// SIMATIC STEP 7 (V5.x) project 1300
// CPU: CPU 315-2 DP
// station: P_ADR_BUS
// station: Hardware
// station: SIMATIC 300(1)
// program: S7 Program(1)

SYMBOL_TABLE
"CLOCK_OP"	DB 5	DB 5	// COMMUNICATION CLOCK OP
"TransferValves"	DB 10	DB 10	// Data Transfer for Valves
"TransferMotor"	DB 11	DB 11	// Data Transfer for Motor
"TransferLevel"	DB 12	DB 12	// Data Transfer for Level
"TransferPressure"	DB 13	DB 13	// Data Transfer for Pressure
"TransferTemperature"	DB 14	DB 14	// Data Transfer for Temperatuer
"TransferPID"	DB 15	DB 15	// Data Transfer for PID
"TransferFlow"	DB 16	DB 16	// Data Transfer for Flow
"TrasferViskosity"	DB 17	DB 17	// Data Transfer for Viskosity
"TransferWeight"	DB 18	DB 18	// Data Transfer for Weight
"TransferGenerell"	DB 30	DB 30	// Data Transfer Generell
"Instance_FC_9_00"	DB 50	FB 110	// Instancename
"Instance_TC_10_01"	DB 51	FB 110	// Instance TC 10.01
"TransferRecipe"	DB 90	DB 90	// Data Transfer fo Recipe
"TransferBatch"	DB 91	DB 91
"DataBatchStarch"	DB 92	FB 90
"DataBatchCaCO3"	DB 93	FB 90
"ALARMTIME"	DB 100	DB 100	// actual timers alarms
"ALARMBLOCK"	DB 110	DB 110	// alarm indication to OP
"ALARM_ACK_OP"	DB 115	DB 115	// alarm acknowledge from OP
"LAMPS_ACK"	DB 120	DB 120	// lamp acknowledge
"CLOCK_FB"	FB 5	FB 5	// SETTING CPU CLOCK
"preparation starch"	FB 10	FB 10	// starch preparation
"starch cooking"	FB 11	FB 11	// starch jet cooker
"preparation CaCO3"	FB 15	FB 15	// CaCO3 preparation
"Devices"	FB 20	FB 20	// Devices
"ALARM_HANDLING_STARCH"	FB 31	FB 31	// alarm handling starch
"ALARM_HANDLING_CaCO3"	FB 32	FB 32	// alarm handling CaCO3
"ALARM"	FB 33	FB 33	// indication alarm
"CONT_C"	FB 41	FB 41	// Continuous Control
"Batch"	FB 90	FB 90	// Batch
"Control"	FB 110	FB 110	// Controler
"BatchControlStarch"	FC 10	FC 10	// Batch Control Starch
"BatchControlCaCO3"	FC 11	FC 11	// Batch Control CaCO3
"Recipe Control"	FC 90	FC 90	// Recipe Control
"DosLine"	FC 91	FC 91	// Dosing Line
"AUTO_VALVE"	FC 100	FC 100	// automatic valve
"MOTOR"	FC 101	FC 101	// motor control
"level"	FC 107	FC 107	// level display
"temperature"	FC 109	FC 109	// temperature display
"flow"	FC 110	FC 110	// flow display
"AI_4-20"	FC 111	FC 111	// analog input 4-20mA
"AO_4-20"	FC 112	FC 112	// analog output 4-20mA
"weight"	FC 114	FC 114	// weighing unit
"ALARM_BLOCK"	FC 115	FC 115	// alarm function block
"M2_01_RUN"	I 8.0	BOOL	// screw conveyor cat. Starch running
"M3_01_RUN"	I 8.1	BOOL	// dedusting station cat. Starch running
"M4_01_RUN"	I 8.2	BOOL	// agitator make down tank cat. Starch running
"M5_01_RUN"	I 8.3	BOOL	// agitator storage tank cat. Starch running
"M6_01_RUN"	I 8.4	BOOL	// pump cat. Starch running
"M7_01_RUN"	I 8.5	BOOL	// stby pump cat. Starch running
"M32_01_RUN"	I 8.6	BOOL	// screw conveyor CaCO3 running
"M33_01_RUN"	I 8.7	BOOL	// dedusting station CaCO3 running
"M34_01_RUN"	I 9.0	BOOL	// agitator make down tank CaCO3 running
"HS2_02_ZSC"	I 12.0	BOOL	// valve screw conveyor cat. Starch closed
"HS2_02_ZSO"	I 12.1	BOOL	// valve screw conveyor cat. Starch open
"HS4_05_ZSC"	I 12.2	BOOL	// water valve m.d. tank cat. Starch closed
"HS4_06_ZSC"	I 12.3	BOOL	// discharge valve m.d. tank cat. Starch closed
"HS5_04_ZSC"	I 12.4	BOOL	// disch. valve storage tank cat. Starch closed
"HS6_07_ZSC"	I 12.5	BOOL	// flush valve pump cat. Starch closed
"FS11_00_IN"	I 12.6	BOOL	// flow > minimum dilution water cat. Ctarch
"HS11_01_ZSC"	I 12.7	BOOL	// valve dilution water cat. Starch closed
"HS32_02_ZSC"	I 13.0	BOOL	// valve screw conveyor CaCO3 closed
"HS32_02_ZSO"	I 13.1	BOOL	// valve screw conveyor CaCO3 open
"HS34_05_ZSC"	I 13.2	BOOL	// water valve m.d. tank CaCO3 closed
"HS34_06_ZSC"	I 13.3	BOOL	// discharge valve m.d. tank CaCO3 closed
"XS13_02_K1"	I 13.4	BOOL	// release filling storage tank cat. Starch
"XS13_03_K1"	I 13.5	BOOL	// release filling storage tank CaCO3
"HS4_07_ZSC"	I 13.6	BOOL	// drain valve m.d. tank cat. Starch closed
"HS34_07_ZSC"	I 13.7	BOOL	// drain valve m.d. tank CaCO3 closed
"Signal_0"	M 1.0	BOOL	// Signal 0
"Signal_1"	M 1.1	BOOL	// Signal 1
"1_second"	M 1.2	BOOL	// second pulse
"PB_LAMP_ACK"	M 1.3	BOOL	// Lamp acknowledge
"spike_ pulse_ 1H"	M 2.0	BOOL	// spike pulse 1 houre
"Release_Time"	M 2.1	BOOL	// release timetransfer
"Pulse_Time"	M 2.2	BOOL	// pulse timetransfer
"OP_COMM_OK"	M 9.0	BOOL	// Op Communication ok
"LB_OP_PULS"	M 9.1	BOOL	// Lifebit OP Communikation
"fault_M_2_01"	M 12.0	BOOL	// fault motor M 2.01
"fault_M_3_01"	M 12.1	BOOL	// fault motor M 3.01
"fault_M_4_01"	M 12.2	BOOL	// fault motor M 4.01
"fault_M_5_01"	M 12.3	BOOL	// fault motor M 5.01
"fault_M_6_01"	M 12.4	BOOL	// fault motor M 6.01
"fault_M_7_01"	M 12.5	BOOL	// fault motor M 7.01
"fault_M_32_01"	M 12.6	BOOL	// fault motor M 32.01
"fault_M_33_01"	M 12.7	BOOL	// fault motor M 33.01
"fault_M_34_01"	M 13.0	BOOL	// fault motor M 34.01
"fault_HS_2_02"	M 14.0	BOOL	// fault valve HS 2.02
"fault_HS_2_05"	M 14.1	BOOL	// fault valve HS 2.05
"fault_HS_4_05"	M 14.2	BOOL	// fault valve HS 4.05
"fault_HS_4_06"	M 14.3	BOOL	// fault valve HS 4.06
"fault_HS_4_07"	M 14.4	BOOL	// fault valve HS 4.07
"fault_HS_5_04"	M 14.5	BOOL	// fault valve HS 5.04
"fault_HS_6_07"	M 14.6	BOOL	// fault valve HS 6.07
"fault_HS_11_01"	M 14.7	BOOL	// fault valve HS 11.01
"fault_HS_32_02"	M 15.0	BOOL	// fault valve HS 32.02
"fault_HS_32_05"	M 15.1	BOOL	// fault valve HS 32.05
"fault_HS_34_05"	M 15.2	BOOL	// fault valve HS 34.05
"fault_HS_34_06"	M 15.3	BOOL	// fault valve HS 34.06
"fault_HS_34_07"	M 15.4	BOOL	// fault valve HS 34.07
"fault_WQ_4_04"	M 16.0	BOOL	// fault weighing unit WQ 4.04
"fault_LI_5_03"	M 16.1	BOOL	// fault level transmitter LI 5.03
"fault_FC_9_00"	M 16.2	BOOL	// fault flow transmitter FC 9.00
"fault_TC_10_01"	M 16.3	BOOL	// fault temperature transmitter TC 10.01
"fault_XS_13_02"	M 16.4	BOOL	// fault level transmitter XS 13.02
"fault_WQ_34_04"	M 16.5	BOOL	// fault weighing unit WQ 34.04
"fault_XS_13_03"	M 16.6	BOOL	// fault level transmitter XS 13.03
"fault_FS_11_00"	M 17.0	BOOL	// fault flow FS 11.00
"fault_HH_WQ_4_04"	M 18.0	BOOL	// fault Alarm maximum WQ 4.04
"fault_HH_LI_5_03"	M 18.1	BOOL	// fault Alarm maximum LI 5.03
"fault_HH_FC_9_00"	M 18.2	BOOL	// fault Alarm maximum FC 9.00
"fault_LL_FC_9_00"	M 18.3	BOOL	// fault Alarm minimum FC 9.00
"fault_HH_TC_10_01"	M 18.4	BOOL	// fault Alarm maximum TC 10.01
"fault_LL_TC_10_01"	M 18.5	BOOL	// fault Alarm minimum TC 10.01
"fault_HH_XS_13_02"	M 18.6	BOOL	// fault Alarm maximum XS 13.02
"fault_LL_XS_13_02"	M 18.7	BOOL	// fault Alarm minimum XS 13.02
"fault_HH_WQ_34_04"	M 19.0	BOOL	// fault Alarm maximum WQ 34.04
"fault_HH_XS_13_03"	M 19.1	BOOL	// fault Alarm maximum XS 13.03
"fault_LL_XS_13_03"	M 19.2	BOOL	// fault Alarm minimum XS 13.03
"HH_WQ_4_04"	M 60.0	BOOL	// Alarm HH weighing unit WQ 4.04
"HH_LI_5_03"	M 60.1	BOOL	// Alarm HH level transmitter LI 5.03
"HH_FC_9_00"	M 60.2	BOOL	// Alarm HH flow transmitter FC 9.00
"HH_TC_10_01"	M 60.3	BOOL	// Alarm HH temperature transmitter TC 10.01
"HH_XS_13_02"	M 60.4	BOOL	// Alarm HH level transmitter XS 13.02
"HH_WQ_34_04"	M 60.5	BOOL	// Alarm HH weighing unit WQ 34.04
"HH_XS_13_03"	M 60.6	BOOL	// Alarm HH level transmitter XS 13.03
"H_WQ_4_04"	M 61.0	BOOL	// Alarm H weighing unit WQ 4.04
"H_LI_5_03"	M 61.1	BOOL	// Alarm H level transmitter LI 5.03
"H_FC_9_00"	M 61.2	BOOL	// Alarm H flow transmitter FC 9.00
"H_TC_10_01"	M 61.3	BOOL	// Alarm H temperature transmitter TC 10.01
"H_XS_13_02"	M 61.4	BOOL	// Alarm H level transmitter XS 13.02
"H_WQ_34_04"	M 61.5	BOOL	// Alarm H weighing unit WQ 34.04
"H_XS_13_03"	M 61.6	BOOL	// Alarm H level transmitter XS 13.03
"L_WQ_4_04"	M 62.0	BOOL	// Alarm L weighing unit WQ 4.04
"L_LI_5_03"	M 62.1	BOOL	// Alarm L level transmitter LI 5.03
"L_FC_9_00"	M 62.2	BOOL	// Alarm L flow transmitter FC 9.00
"L_TC_10_01"	M 62.3	BOOL	// Alarm L temperature transmitter TC 10.01
"L_XS_13_02"	M 62.4	BOOL	// Alarm L level transmitter XS 13.02
"L_WQ_34_04"	M 62.5	BOOL	// Alarm L weighing unit WQ 34.04
"L_XS_13_03"	M 62.6	BOOL	// Alarm L level transmitter XS 13.03
"LL_WQ_4_04"	M 63.0	BOOL	// Alarm LL weighing unit WQ 4.04
"LL_LI_5_03"	M 63.1	BOOL	// Alarm LL Level transmitter LLI 5.03
"LL_FC_9_00"	M 63.2	BOOL	// Alarm LL flow transmitter FC 9.00
"LL_TC_10_01"	M 63.3	BOOL	// Alarm LL temperature transmitter TC 10.01
"LL_XS_13_02"	M 63.4	BOOL	// Alarm LL Level transmitter XS 13.02
"LL_WQ_34_04"	M 63.5	BOOL	// Alarm LL weighing unit WQ 34.04
"LL_XS_13_03"	M 63.6	BOOL	// Alarm LL Level transmitter XS 13.03
"check_M_2_01"	M 70.0	BOOL	// check motor M 2.01
"check_M_3_01"	M 70.1	BOOL	// check motor M 3.01
"check_M_4_01"	M 70.2	BOOL	// check motor M 4.01
"check_M_5_01"	M 70.3	BOOL	// check motor M 5.01
"check_M_6_01"	M 70.4	BOOL	// check motor M 6.01
"check_M_7_01"	M 70.5	BOOL	// check motor M 7.01
"check_M_32_01"	M 70.6	BOOL	// check motor M 32.01
"check_M_33_01"	M 70.7	BOOL	// check motor M 33.01
"check_M_34_01"	M 71.0	BOOL	// check motor M 34.01
"check_HS_2_02"	M 72.0	BOOL	// check valve HS 2.02
"check_HS_2_05"	M 72.1	BOOL	// check valve HS 2.05
"check_HS_4_05"	M 72.2	BOOL	// check valve HS 4.05
"check_HS_4_06"	M 72.3	BOOL	// check valve HS 4.06
"check_HS_4_07"	M 72.4	BOOL	// check valve HS 4.07
"check_HS_5_04"	M 72.5	BOOL	// check valve HS 5.04
"check_HS_6_07"	M 72.6	BOOL	// check valve HS 6.07
"check_HS_11_01"	M 72.7	BOOL	// check valve HS 11.01
"check_HS_32_02"	M 73.0	BOOL	// check valve HS 32.02
"check_HS_32_05"	M 73.1	BOOL	// check valve HS 32.05
"check_HS_34_05"	M 73.2	BOOL	// check valve HS 34.05
"check_HS_34_06"	M 73.3	BOOL	// check valve HS 34.06
"check_HS_34_07"	M 73.4	BOOL	// check valve HS 34.07
"check_WQ_4_04"	M 74.0	BOOL	// check weighing unit WQ 4.04
"check_LI_5_03"	M 74.1	BOOL	// check Level transmitter LLI 5.03
"check_FC_9_00"	M 74.2	BOOL	// check flow transmitter FC 9.00
"check_TC_10_01"	M 74.3	BOOL	// check temperature transmitter TC 10.01
"check_XS_13_02"	M 74.4	BOOL	// check Level transmitter XS 13.02
"check_WQ_34_04"	M 74.5	BOOL	// check weighing unit WQ 34.04
"check_XS_13_03"	M 74.6	BOOL	// check Level transmitter XS 13.03
"check_FS_11_00"	M 75.0	BOOL	// check flow FS 11.00
"fault_ack_M_2_01"	M 90.0	BOOL	// fault acknowledge motor M 2.01
"fault_ack_M_3_01"	M 90.1	BOOL	// fault acknowledge motor M 3.01
"fault_ack_M_4_01"	M 90.2	BOOL	// fault acknowledge motor M 4.01
"fault_ack_M_5_01"	M 90.3	BOOL	// fault acknowledge motor M 5.01
"fault_ack_M_6_01"	M 90.4	BOOL	// fault acknowledge motor M 6.01
"fault_ack_M_7_01"	M 90.5	BOOL	// fault acknowledge motor M 7.01
"fault_ack_M_32_01"	M 90.6	BOOL	// fault acknowledge motor M 32.01
"fault_ack_M_33_01"	M 90.7	BOOL	// fault acknowledge motor M 33.01
"fault_ack_M_34_01"	M 91.0	BOOL	// fault acknowledge motor M 34.01
"fault_ack_HS_2_02"	M 92.0	BOOL	// fault acknowledge valve HS 2.02
"fault_ack_HS_2_05"	M 92.1	BOOL	// fault acknowledge valve HS 2.05
"fault_ack_HS_4_05"	M 92.2	BOOL	// fault acknowledge valve HS 4.05
"fault_ack_HS_4_06"	M 92.3	BOOL	// fault acknowledge valve HS 4.06
"fault_ack_HS_4_07"	M 92.4	BOOL	// fault acknowledge valve HS 4.07
"fault_ack_HS_5_04"	M 92.5	BOOL	// fault acknowledge valve HS 5.04
"fault_ack_HS_6_07"	M 92.6	BOOL	// fault acknowledge valve HS 6.07
"fault_ack_HS_11_01"	M 92.7	BOOL	// fault acknowledge valve HS 11.01
"fault_ack_HS_32_02"	M 93.0	BOOL	// fault acknowledge valve HS 32.02
"fault_ack_HS_32_05"	M 93.1	BOOL	// fault acknowledge valve HS 32.05
"fault_ack_HS_34_05"	M 93.2	BOOL	// fault acknowledge valve HS 34.05
"fault_ack_HS_34_06"	M 93.3	BOOL	// fault acknowledge valve HS 34.06
"fault_ack_HS_34_07"	M 93.4	BOOL	// fault acknowledge valve HS 34.07
"fault_ack_WQ_4_04"	M 94.0	BOOL	// fault acknowledge weighing unit WQ 4.04
"fault_ack_LI_5_03"	M 94.1	BOOL	// fault acknowledge Level transmitter LLI 5.03
"fault_ack_FC_9_00"	M 94.2	BOOL	// fault acknowledge flow transmitter FC 9.00
"fault_ack_TC_10_01"	M 94.3	BOOL	// fault acknowledge temperature transmitter TC 10.01
"fault_ack_XS_13_02"	M 94.4	BOOL	// fault acknowledge Level transmitter XS 13.02
"fault_ack_WQ_34_04"	M 94.5	BOOL	// fault acknowledge weighing unit WQ 34.04
"fault_ack_XS_13_03"	M 94.6	BOOL	// fault acknowledge Level transmitter XS 13.03
"fault_ack_FS_11_00"	M 95.0	BOOL	// fault acknowledge flow FS 11.00
"fault_ack_HH_WQ_4_04"	M 96.0	BOOL	// fault acknowledge Alarm maximum WQ 4.04
"fault_ack_HH_LI_5_03"	M 96.1	BOOL	// fault acknowledge Alarm maximum LI 5.03
"fault_ack_HH_FC_9_00"	M 96.2	BOOL	// fault acknowledge Alarm maximum FC 9.00
"fault_ack_LL_FC_9_00"	M 96.3	BOOL	// fault acknowledge Alarm minimum FC 9.00
"fault_ack_HH_TC_10_01"	M 96.4	BOOL	// fault acknowledge Alarm maximum TC 10.01
"fault_ack_LL_TC_10_01"	M 96.5	BOOL	// fault acknowledge Alarm minimum TC 10.01
"fault_ack_HH_XS_13_02"	M 96.6	BOOL	// fault acknowledge Alarm maximum XS 13.02
"fault_ack_LL_XS_13_02"	M 96.7	BOOL	// fault acknowledge Alarm minimum XS 13.02
"fault_ack_HH_WQ_34_04"	M 97.0	BOOL	// fault acknowledge Alarm maximum WQ 34.04
"fault_ack_HH_XS_13_03"	M 97.1	BOOL	// fault acknowledge Alarm maximum XS 13.03
"fault_ack_LL_XS_13_03"	M 97.2	BOOL	// fault acknowledge Alarm minimum XS 13.03
"auto_on_M_2_01"	M 100.0	BOOL	// auto on motor M 2.01
"auto_on_M_3_01"	M 100.1	BOOL	// auto on motor M 3.01
"auto_on_M_4_01"	M 100.2	BOOL	// auto on motor M 4.01
"auto_on_M_5_01"	M 100.3	BOOL	// auto on motor M 5.01
"auto_on_M_6_01"	M 100.4	BOOL	// auto on motor M 6.01
"auto_on_M_7_01"	M 100.5	BOOL	// auto on motor M 7.01
"auto_on_M_32_01"	M 100.6	BOOL	// auto on motor M 32.01
"auto_on_M_33_01"	M 100.7	BOOL	// auto on motor M 33.01
"auto_on_M_34_01"	M 101.0	BOOL	// auto on motor M 34.01
"auto_on_HS_2_02"	M 102.0	BOOL	// auto on valve HS 2.02
"auto_on_HS_2_05"	M 102.1	BOOL	// auto on valve HS 2.05
"auto_on_HS_4_05"	M 102.2	BOOL	// auto on valve HS 4.05
"auto_on_HS_4_06"	M 102.3	BOOL	// auto on valve HS 4.06
"auto_on_HS_4_07"	M 102.4	BOOL	// auto on valve HS 4.07
"auto_on_HS_5_04"	M 102.5	BOOL	// auto on valve HS 5.04
"auto_on_HS_6_07"	M 102.6	BOOL	// auto on valve HS 6.07
"auto_on_HS_11_01"	M 102.7	BOOL	// auto on valve HS 11.01
"auto_on_HS_32_02"	M 103.0	BOOL	// auto on valve HS 32.02
"auto_on_HS_32_05"	M 103.1	BOOL	// auto on valve HS 32.05
"auto_on_HS_34_05"	M 103.2	BOOL	// auto on valve HS 34.05
"auto_on_HS_34_06"	M 103.3	BOOL	// auto on valve HS 34.06
"auto_on_HS_34_07"	M 103.4	BOOL	// auto on valve HS 34.07
"imp_flush_start"	M 103.5	BOOL	// impuls flushing start starch
"Cond_Dos_Starch"	M 120.0	BOOL	// Condition Dosing Starch
"Agitator_Stop_Starch"	M 120.2	BOOL	// Condition Agitator Stop Starch
"Save_Dis_On_Starch"	M 120.3	BOOL	// Save discharge was on starch
"Cond_Dos_CaCO3"	M 121.0	BOOL	// Condition Dosing CaCO3
"Agitator_Stop_CaCO3"	M 121.2	BOOL	// Condition Stop Agitator CaCO3
"Save_Dis_On_CaCO3"	M 121.3	BOOL	// Save discharge was on CaCO3
"Devices_auto_Starch"	M 130.0	BOOL	// Devices automatic mode starch
"fault_starch_cooking"	M 130.1	BOOL	// fault Starch cooking
"cooking_on_starch"	M 130.2	BOOL	// Cooking on starch
"cooking_end_starch"	M 130.3	BOOL	// cooking end starch
"cond_flushig_starch"	M 130.4	BOOL	// condition flushing starch
"SlurryStorageEmptyStarch"	M 130.5	BOOL	// Slurry Storage Tank empty Starch
"flushing_on_starch"	M 130.6	BOOL	// flushing on starch
"Pulse_Force_Flow_Start"	M 137.0	BOOL	// Pulse force start flow starch cooking
"Pulse_Force_Flow_Flush"	M 137.1	BOOL	// Pulse force flushing flow starch cooking
"Force_Flow_On_Starch"	M 137.2	BOOL	// Force flow on starch cooking
"Pump_auto_running_starch"	M 137.3	BOOL	// pump running auto mode
"Coinz_Prod_Steam_Valve"	M 137.4	BOOL	// Coinz Product to Steam Valve
"Force_Steam_On_Starch"	M 137.5	BOOL	// Force steam on starch cooking
"Force_Steam_Off_Starch"	M 137.6	BOOL	// Force steam off starch cooking
"LL_Alarm_Flush_Starch"	M 137.7	BOOL	// Alarm LL Flushing starch
"PulseFlushOn"	M 138.0	BOOL	// Impulse flushing on
"Coinz_Prod_Dilution"	M 138.1	BOOL	// Coinz Product to Dilution Station
"Coinz_Water_Steam_Valve"	M 138.2	BOOL	// Coinz Water to Steamvalve
"Coinz_Water_Dilution"	M 138.3	BOOL	// Coinz Water to Dilution Station
"Coinz_Water_Pipe"	M 138.4	BOOL	// Coinz Water in pipe
"PulseCoinzDilutionOn"	M 138.5	BOOL	// Impulse coinz product to Dilution Station
"IMP_START_STARCH"	M 160.0	BOOL	// Impuls Start Batch Starch
"Hold_Mixing_Time_Starch"	M 160.1	BOOL	// Hold Mixing Time Starch
"Discharged1_Starch"	M 161.0	BOOL	// Discharged 1 starch
"Discharged2_Starch"	M 161.1	BOOL	// Discharged 2 starch
"Batch_Starch_Running"	M 180.0	BOOL	// Batch Starch Running
"Batch_Starch_Started"	M 180.1	BOOL	// Batch Starch Started
"Dos_On_Water_Starch"	M 185.0	BOOL	// Dosing on water starch
"Cmd_Agitator_On_Starch"	M 185.1	BOOL	// Command Agitator on starch
"Dos_On_Powder_Starch"	M 185.2	BOOL	// Dosing on powder starch
"Cmd_Discharge1_On_Starch"	M 185.3	BOOL	// Command discharge 1 on starch
"Active_Discharge1_Starch"	M 185.4	BOOL	// Active Discharge 1 Starch
"Dos_On_Flushwater_Starch"	M 185.5	BOOL	// Dosing on flushwater starch
"Cmd_Discharge2_On_Starch"	M 185.6	BOOL	// Command discharge 2 on starch
"Active_Discharge2_Starch"	M 185.7	BOOL	// Active Discharge 2 Starch
"IMP_START_CaCO3"	M 190.0	BOOL	// Impuls Start Batch CaCO3
"Hold_Mixing_Time_CaCO3"	M 190.1	BOOL	// Hold Mixing Time CaCO3
"Discharged1_CaCO3"	M 191.0	BOOL	// Discharged 1 CaCO3
"Discharged2_CaCO3"	M 191.1	BOOL	// Discharged 2 CaCO3
"Batch_CaCO3_Running"	M 210.0	BOOL	// Batch CaCO3 Running
"Batch_CaCO3_Started"	M 210.1	BOOL	// Batch CaCO3 Started
"Dos_On_Water_CaCO3"	M 215.0	BOOL	// Dosing on water CaCO3
"Cmd_Agitator_On_CaCO3"	M 215.1	BOOL	// Command Agitator on CaCO3
"Dos_On_Powder_CaCO3"	M 215.2	BOOL	// Dosing on powder CaCO3
"Cmd_Discharge1_On_CaCO3"	M 215.3	BOOL	// Command discharge 1 on CaCO3
"Active_Discharge1_CaCO3"	M 215.4	BOOL	// Active Discharge 1 CaCO3
"Dos_On_Flushwater_CaCO3"	M 215.5	BOOL	// Dosing on flushwater CaCO3
"Cmd_Discharge2_On_CaCO3"	M 215.6	BOOL	// Command discharge 2 on CaCO3
"Active_Discharge2_CaCO3"	M 215.7	BOOL	// Active Discharge 2 CaCO3
"WQ_4_04_Value"	MD 30	REAL	// value WQ 4.04
"WQ_34_04_Value"	MD 34	REAL	// value WQ 34.04
"LI_5_03_Percent"	MD 38	REAL	// percent LI 5.03
"FC_9_00_Value"	MD 42	REAL	// value FC 9.00
"TC_10_01_Value"	MD 46	REAL	// value TC 10.01
"XS_13_02_Percent"	MD 50	REAL	// percent XS 13.02
"XS_13_03_Percent"	MD 54	REAL	// percent XS 13.03
"ActVolumePumps"	MD 220	REAL	// Actual Volume pumps
"ActValueSlurryMinStarch"	MD 224	REAL	// Actual Value Slurry under minimum
"Cycle_Time"	MW 252	INT	// Cycle Time
"MOD_ERR"	OB 122	OB 122	// Module Access Error
"LI5_02_IN"	PIW 256	WORD	// level storage tank cat. starch
"TT10_01_IN"	PIW 258	WORD	// temperature control cat. starch cooker
"WQ4_04_IN"	PIW 260	WORD	// weight make down tank cat. starch
"FC9_00_IN"	PIW 262	WORD	// flow control cat. starch
"PI10_13_IN"	PIW 264	WORD	// pressure indication jet cooker
"WQ34_04_IN"	PIW 266	WORD	// weight make down tank CaCO3
"XS13_02_LI"	PIW 268	WORD	// level storage tank cooked cat. starch
"XS13_03_LI"	PIW 270	WORD	// level storage tank cooked CaCO3
"SC6_01_SET"	PQW 272	WORD	// speed control pump cat. starch
"SC7_02_SET"	PQW 274	WORD	// speed control stby pump cat. starch
"TV10_02_OUT"	PQW 276	WORD	// temperature control cat. starch cooker
"M2_01_ON"	Q 16.0	BOOL	// screw conveyor cat. Starch on
"M3_01_ON"	Q 16.1	BOOL	// dedusting station cat. Starch on
"M3_01_ST"	Q 16.2	BOOL	// dedusting station cat. Starch on
"M4_01_ON"	Q 16.3	BOOL	// agitator make down tank cat. Starch on
"M5_01_ON"	Q 16.4	BOOL	// agitator storage tank cat. Starch on
"M6_01_ON"	Q 16.5	BOOL	// pump cat. Starch on
"M7_01_ON"	Q 16.6	BOOL	// stby pump cat. Starch on
"HS2_02_ON"	Q 16.7	BOOL	// valve screw conveyor cat. Starch on
"HS4_05_ON"	Q 17.0	BOOL	// water valve m.d. tank cat. Starch on
"HS4_06_ON"	Q 17.1	BOOL	// discharge valve m.d. tank cat. Starch on
"HS5_04_ON"	Q 17.2	BOOL	// disch. valve storage tank cat. Starch on
"HS6_07_ON"	Q 17.3	BOOL	// flush valve pump cat. Starch on
"HS11_01_ON"	Q 17.4	BOOL	// valve dilution water cat. Starch on
"HS32_02_ON"	Q 17.5	BOOL	// valve screw conveyor CaCO3 on
"HS34_05_ON"	Q 17.6	BOOL	// water valve m.d. tank CaCO3 on
"HS34_06_ON"	Q 17.7	BOOL	// discharge valve m.d. tank CaCO3 on
"M32_01_ON"	Q 20.0	BOOL	// screw conveyor CaCO3 on
"M33_01_ON"	Q 20.1	BOOL	// dedusting station CaCO3 on
"M33_01_ST"	Q 20.2	BOOL	// dedusting station CaCO3 valve on
"M34_01_ON"	Q 20.3	BOOL	// agitator make down tank CaCO3 on
"XA13_01_ON"	Q 20.4	BOOL	// alarm preparation
"XS13_02_K2"	Q 20.5	BOOL	// filling is on storage tank cat. starch
"XS13_02_K3"	Q 20.6	BOOL	// fault filling storage tank cat. starch
"XS13_03_K2"	Q 20.7	BOOL	// filling is on storage tank CaCO3
"XS13_03_K3"	Q 21.0	BOOL	// fault filling storage tank CaCO3
"HS2_05_ON"	Q 21.1	BOOL	// air valve screw conveyor cat. Starch on
"HS4_07_ON"	Q 21.2	BOOL	// drain valve m.d. tank cat. Starch on
"HS32_05_ON"	Q 21.3	BOOL	// air valve screw conveyor CaCO3 on
"HS34_07_ON"	Q 21.4	BOOL	// drain valve m.d. tank CaCO3 on
"TON"	SFB 4	SFB 4	// Generate an On Delay
"SET_CLK"	SFC 0	SFC 0	// Set System Clock
"Valve UDT"	UDT 1	UDT 1	// Data Valve
"Valve Popup UDT"	UDT 2	UDT 2	// Data Valve Popup
"Motor UDT"	UDT 3	UDT 3	// Data Motor
"Motor Popup UDT"	UDT 4	UDT 4	// Data Motor Popup
"Level UDT"	UDT 5	UDT 5	// Data Level
"Level Popup UDT"	UDT 6	UDT 6	// Data Level Popup
"Pressure UDT"	UDT 7	UDT 7	// Data Pressure
"Pressure Popup UDT"	UDT 8	UDT 8	// Data Pressure Popup
"Temperature UDT"	UDT 9	UDT 9	// Data Temperature
"Temperature Popup UDT"	UDT 10	UDT 10	// Data Temperature Popup
"Controler UDT"	UDT 11	UDT 11	// Data Controler
"Controler Popup UDT"	UDT 12	UDT 12	// Data Controler Popup
"Flow UDT"	UDT 13	UDT 13	// Data Flow
"Flow Popup UDT"	UDT 14	UDT 14	// Data Flow Popup
"Viskosity UDT"	UDT 15	UDT 15	// Viskosity Data
"Viskosity Popup UDT"	UDT 16	UDT 16	// Data Viskosity Popup
"Weight UDT"	UDT 17	UDT 17	// Weight Data
"Weight Popup UDT"	UDT 18	UDT 18	// Data Weight Popup
"Recipe UDT"	UDT 90	UDT 90	// Data Recipe
"DosLine UDT"	UDT 91	UDT 91	// Dosing Line UDT
"VAT_1"	VAT 1	
END_SYMBOL_TABLE

FUNCTION_BLOCK "CLOCK_FB"	// FB 5
AUTHOR : gaw-be
FAMILY : GAW
NAME : DATETIME
VERSION : 0.1
BEGIN
// (block stored without names or comments; labels and parameter names are numbered)
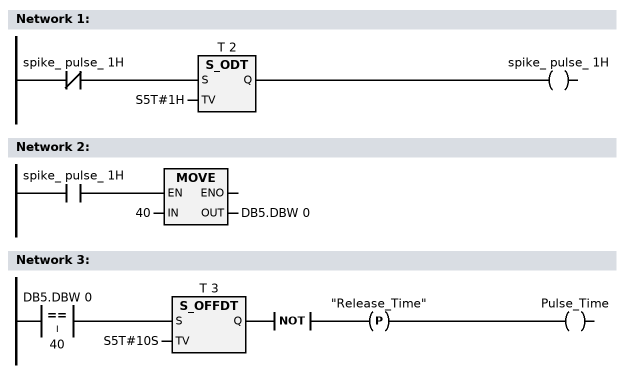
NETWORK
TITLE =
      AN    "spike_ pulse_ 1H";
      L     S5T#1H;
      SD    T 2;
      NOP   0;
      NOP   0;
      NOP   0;
      A     T 2;
      =     "spike_ pulse_ 1H";
NETWORK
TITLE =
      A     "spike_ pulse_ 1H";
      JNB   M001;
      L     40;
      T     DB5.DBW 0;
M001: NOP   0;
NETWORK
TITLE =
      A(;
      A(;
      L     DB5.DBW 0;
      L     40;
      ==I;
      );
      L     S5T#10S;
      SF    T 3;
      NOP   0;
      NOP   0;
      NOP   0;
      A     T 3;
      );
      NOT;
      FP    "Release_Time";
      =     "Pulse_Time";
NETWORK
TITLE =
      A     "Pulse_Time";
      JNB   M002;
      BLD   7;
      L     5;
      T     LW 102;
      L     P#DBX 8.0;
      T     LD 104;
      UC    "SET_CLK";
      {     P#L 102.0, P#L 100.0 };
      BLD   8;
M002: NOP   0;
END_FUNCTION_BLOCK

FUNCTION_BLOCK "preparation starch"	// FB 10
VERSION : 0.1
BEGIN
// (block stored without names or comments; labels and parameter names are numbered)
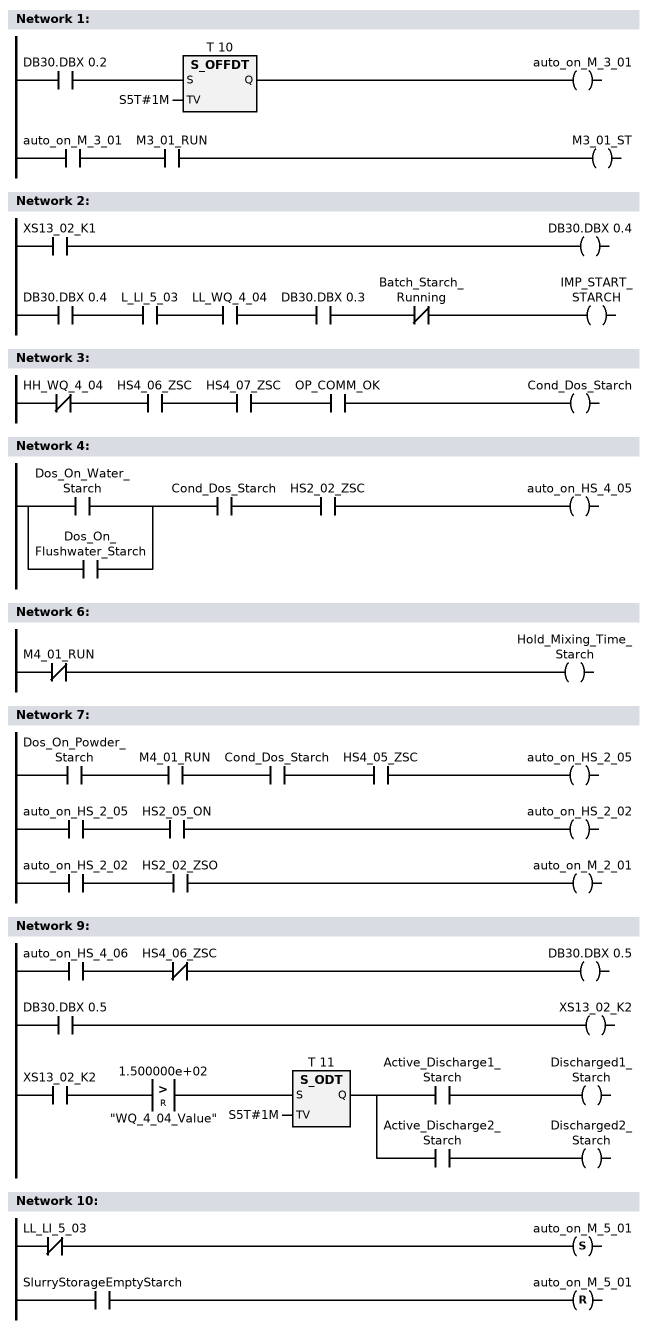
NETWORK
TITLE =
      A(;
      A     DB30.DBX 0.2;
      L     S5T#1M;
      SF    T 10;
      NOP   0;
      NOP   0;
      NOP   0;
      A     T 10;
      );
      =     "auto_on_M_3_01";
      A     "auto_on_M_3_01";
      A     "M3_01_RUN";
      =     "M3_01_ST";
NETWORK
TITLE =
      A     "XS13_02_K1";
      =     DB30.DBX 0.4;
      A     DB30.DBX 0.4;
      A     "L_LI_5_03";
      A     "LL_WQ_4_04";
      A     DB30.DBX 0.3;
      AN    "Batch_Starch_Running";
      =     "IMP_START_STARCH";
NETWORK
TITLE =
      AN    "HH_WQ_4_04";
      A     "HS4_06_ZSC";
      A     "HS4_07_ZSC";
      A     "OP_COMM_OK";
      =     "Cond_Dos_Starch";
NETWORK
TITLE =
      A(;
      O     "Dos_On_Water_Starch";
      O     "Dos_On_Flushwater_Starch";
      );
      A     "Cond_Dos_Starch";
      A     "HS2_02_ZSC";
      =     "auto_on_HS_4_05";
NETWORK
TITLE =
      AN    "LL_WQ_4_04";
      A     "Cmd_Agitator_On_Starch";
      A(;
      A(;
      A     "Cmd_Discharge1_On_Starch";
      A     "L_WQ_4_04";
      S     "Agitator_Stop_Starch";
      AN    "Batch_Starch_Running";
      R     "Agitator_Stop_Starch";
      A     "Agitator_Stop_Starch";
      );
      NOT;
      );
      =     "auto_on_M_4_01";
NETWORK
TITLE =
      AN    "M4_01_RUN";
      =     "Hold_Mixing_Time_Starch";
NETWORK
TITLE =
      A     "Dos_On_Powder_Starch";
      A     "M4_01_RUN";
      A     "Cond_Dos_Starch";
      A     "HS4_05_ZSC";
      =     "auto_on_HS_2_05";
      A     "auto_on_HS_2_05";
      A     "HS2_05_ON";
      =     "auto_on_HS_2_02";
      A     "auto_on_HS_2_02";
      A     "HS2_02_ZSO";
      =     "auto_on_M_2_01";
NETWORK
TITLE =
      A(;
      A(;
      O     "L_LI_5_03";
      O(;
      A     "auto_on_HS_4_06";
      A     "Active_Discharge1_Starch";
      S     "Save_Dis_On_Starch";
      AN    "Active_Discharge1_Starch";
      R     "Save_Dis_On_Starch";
      A     "Save_Dis_On_Starch";
      );
      );
      A     "Cmd_Discharge1_On_Starch";
      A     "Active_Discharge1_Starch";
      O;
      A     "Cmd_Discharge2_On_Starch";
      A     "Active_Discharge2_Starch";
      );
      AN    "HH_LI_5_03";
      =     "auto_on_HS_4_06";
NETWORK
TITLE =
      A     "auto_on_HS_4_06";
      AN    "HS4_06_ZSC";
      =     DB30.DBX 0.5;
      A     DB30.DBX 0.5;
      =     "XS13_02_K2";
      A     "XS13_02_K2";
      A(;
      L     1.500000e+02;
      L     "WQ_4_04_Value";
      >R;
      );
      L     S5T#1M;
      SD    T 11;
      NOP   0;
      NOP   0;
      NOP   0;
      A     T 11;
      =     L 0.0;
      A     L 0.0;
      A     "Active_Discharge1_Starch";
      =     "Discharged1_Starch";
      A     L 0.0;
      A     "Active_Discharge2_Starch";
      =     "Discharged2_Starch";
NETWORK
TITLE =
      AN    "LL_LI_5_03";
      S     "auto_on_M_5_01";
      A     "SlurryStorageEmptyStarch";
      R     "auto_on_M_5_01";
      NOP   0;
END_FUNCTION_BLOCK

FUNCTION_BLOCK "starch cooking"	// FB 11
VERSION : 0.1
BEGIN
// (block stored without names or comments; labels and parameter names are numbered)
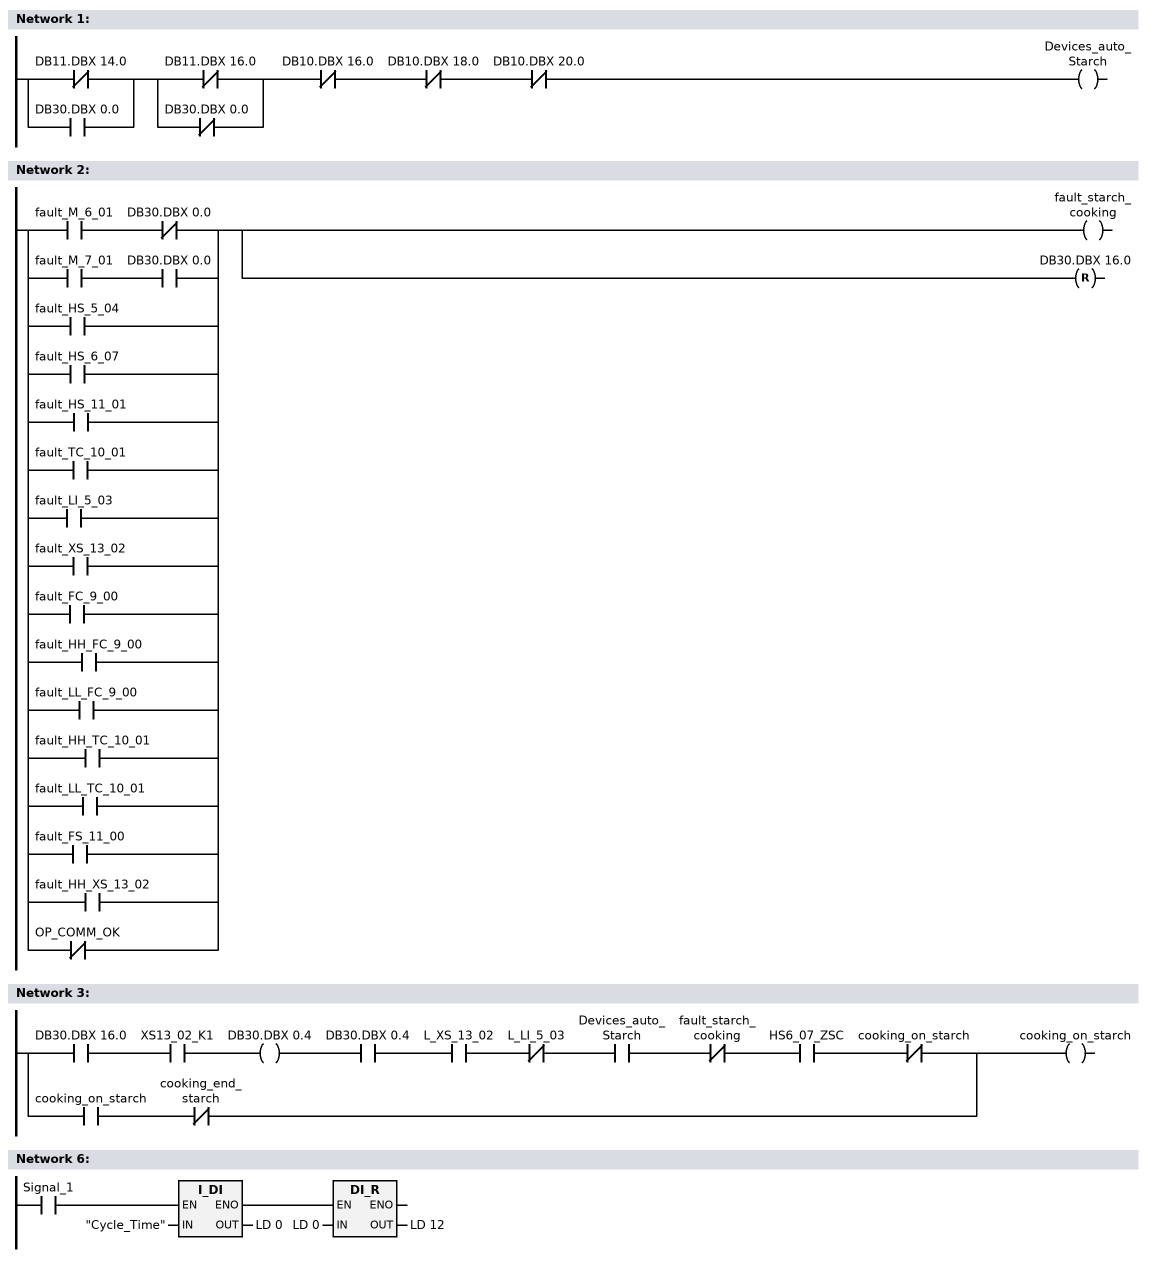
NETWORK
TITLE =
      A(;
      ON    DB11.DBX 14.0;
      O     DB30.DBX 0.0;
      );
      A(;
      ON    DB11.DBX 16.0;
      ON    DB30.DBX 0.0;
      );
      AN    DB10.DBX 16.0;
      AN    DB10.DBX 18.0;
      AN    DB10.DBX 20.0;
      =     "Devices_auto_Starch";
NETWORK
TITLE =
      A     "fault_M_6_01";
      AN    DB30.DBX 0.0;
      O;
      A     "fault_M_7_01";
      A     DB30.DBX 0.0;
      O     "fault_HS_5_04";
      O     "fault_HS_6_07";
      O     "fault_HS_11_01";
      O     "fault_TC_10_01";
      O     "fault_LI_5_03";
      O     "fault_XS_13_02";
      O     "fault_FC_9_00";
      O     "fault_HH_FC_9_00";
      O     "fault_LL_FC_9_00";
      O     "fault_HH_TC_10_01";
      O     "fault_LL_TC_10_01";
      O     "fault_FS_11_00";
      O     "fault_HH_XS_13_02";
      ON    "OP_COMM_OK";
      =     "fault_starch_cooking";
      R     DB30.DBX 16.0;
NETWORK
TITLE =
      A     DB30.DBX 16.0;
      A(;
      A     "XS13_02_K1";
      =     DB30.DBX 0.4;
      A     DB30.DBX 0.4;
      );
      A     "L_XS_13_02";
      AN    "L_LI_5_03";
      A     "Devices_auto_Starch";
      AN    "fault_starch_cooking";
      A     "HS6_07_ZSC";
      AN    "cooking_on_starch";
      O;
      A     "cooking_on_starch";
      AN    "cooking_end_starch";
      =     "cooking_on_starch";
NETWORK
TITLE =
      A(;
      A     "cooking_on_starch";
      AN    "HS5_04_ZSC";
      AN    "cond_flushig_starch";
      S     "cond_flushig_starch";
      A     "cooking_end_starch";
      R     "cond_flushig_starch";
      A     "cond_flushig_starch";
      );
      A(;
      ON    DB30.DBX 16.0;
      ON    "XS13_02_K1";
      O     "H_XS_13_02";
      O     "fault_starch_cooking";
      ON    "Devices_auto_Starch";
      O     "SlurryStorageEmptyStarch";
      );
      S     "flushing_on_starch";
      A     "cooking_end_starch";
      R     "flushing_on_starch";
      NOP   0;
NETWORK
TITLE =
      A(;
      A     "cooking_on_starch";
      A     "HS6_07_ZSC";
      O(;
      A(;
      A     "flushing_on_starch";
      FP    "imp_flush_start";
      L     S5T#10S;
      SF    T 20;
      NOP   0;
      NOP   0;
      NOP   0;
      A     T 20;
      );
      A     "HS6_07_ZSC";
      );
      );
      =     "auto_on_HS_5_04";
      A     "auto_on_HS_5_04";
      AN    "HS5_04_ZSC";
      O(;
      A     "flushing_on_starch";
      A(;
      A(;
      A(;
      A     "LL_FC_9_00";
      A     "auto_on_HS_6_07";
      L     S5T#10S;
      SD    T 24;
      NOP   0;
      NOP   0;
      NOP   0;
      A     T 24;
      );
      S     "LL_Alarm_Flush_Starch";
      AN    "fault_LL_FC_9_00";
      R     "LL_Alarm_Flush_Starch";
      A     "LL_Alarm_Flush_Starch";
      );
      NOT;
      );
      =     "auto_on_HS_6_07";
      A     "auto_on_HS_6_07";
      AN    "HS6_07_ZSC";
      );
      =     L 20.0;
      A     L 20.0;
      AN    DB30.DBX 0.0;
      =     "auto_on_M_6_01";
      A     L 20.0;
      A     DB30.DBX 0.0;
      =     "auto_on_M_7_01";
NETWORK
TITLE =
      A(;
      A     "Signal_1";
      JNB   M001;
      L     "Cycle_Time";
      ITD;
      T     LD 0;
      SET;
      SAVE;
      CLR;
M001: A     BR;
      );
      JNB   M002;
      L     LD 0;
      DTR;
      T     LD 12;
M002: NOP   0;
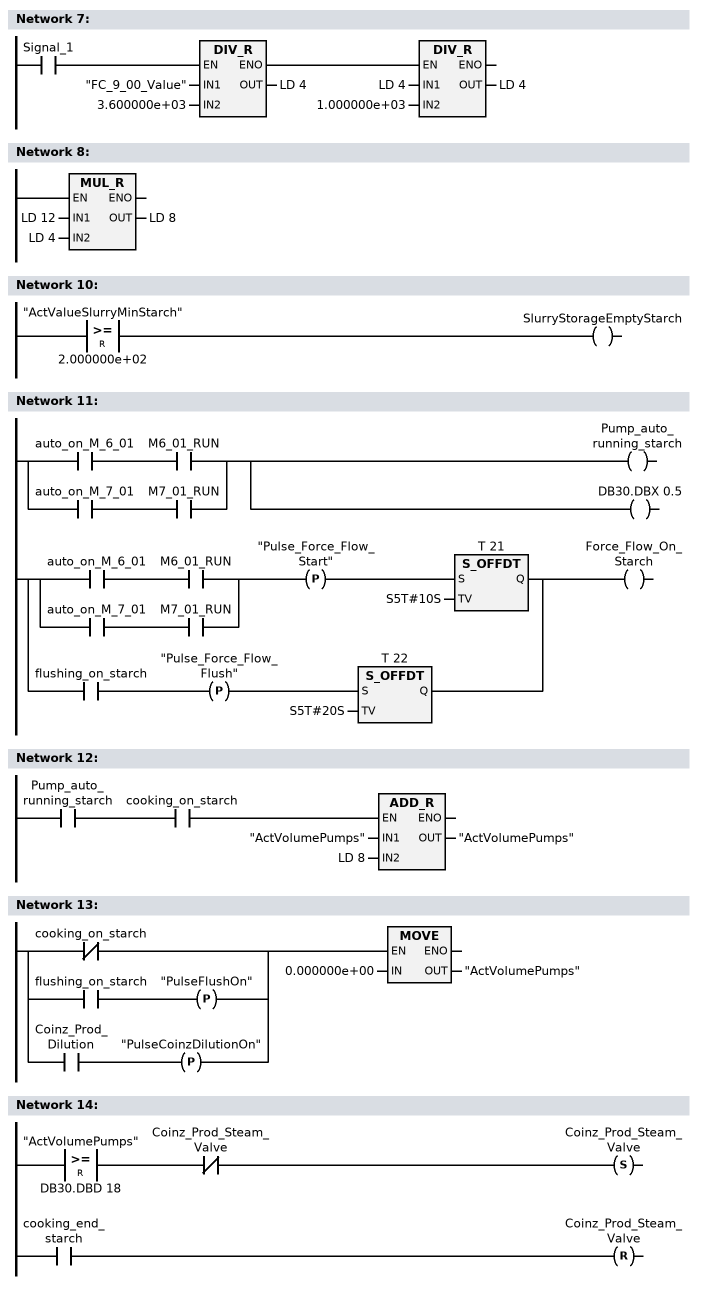
NETWORK
TITLE =
      A(;
      A     "Signal_1";
      JNB   M003;
      L     "FC_9_00_Value";
      L     3.600000e+03;
      /R;
      T     LD 4;
      AN    OV;
      SAVE;
      CLR;
M003: A     BR;
      );
      JNB   M004;
      L     LD 4;
      L     1.000000e+03;
      /R;
      T     LD 4;
M004: NOP   0;
NETWORK
TITLE =
      L     LD 12;
      L     LD 4;
      *R;
      T     LD 8;
      NOP   0;
NETWORK
TITLE =
      L     3.000000e+00;
      L     "LI_5_03_Percent";
      >R;
      =     L 20.0;
      A     "Pump_auto_running_starch";
      A     "auto_on_HS_5_04";
      AN    "HS5_04_ZSC";
      A     L 20.0;
      JNB   M005;
      L     "ActValueSlurryMinStarch";
      L     LD 8;
      +R;
      T     "ActValueSlurryMinStarch";
M005: NOP   0;
      AN    L 20.0;
      JNB   M006;
      L     0.000000e+00;
      T     "ActValueSlurryMinStarch";
M006: NOP   0;
NETWORK
TITLE =
      L     "ActValueSlurryMinStarch";
      L     2.000000e+02;
      >=R;
      =     "SlurryStorageEmptyStarch";
NETWORK
TITLE =
      A     "auto_on_M_6_01";
      A     "M6_01_RUN";
      O;
      A     "auto_on_M_7_01";
      A     "M7_01_RUN";
      =     L 20.0;
      O(;
      A     L 20.0;
      FP    "Pulse_Force_Flow_Start";
      L     S5T#10S;
      SF    T 21;
      NOP   0;
      NOP   0;
      NOP   0;
      A     T 21;
      );
      O(;
      A     "flushing_on_starch";
      FP    "Pulse_Force_Flow_Flush";
      L     S5T#20S;
      SF    T 22;
      NOP   0;
      NOP   0;
      NOP   0;
      A     T 22;
      );
      =     "Force_Flow_On_Starch";
      A     L 20.0;
      BLD   102;
      =     "Pump_auto_running_starch";
      A     L 20.0;
      BLD   102;
      =     DB30.DBX 0.5;
NETWORK
TITLE =
      A     "Pump_auto_running_starch";
      A     "cooking_on_starch";
      JNB   M007;
      L     "ActVolumePumps";
      L     LD 8;
      +R;
      T     "ActVolumePumps";
M007: NOP   0;
NETWORK
TITLE =
      A(;
      ON    "cooking_on_starch";
      O(;
      A     "flushing_on_starch";
      FP    "PulseFlushOn";
      );
      O(;
      A     "Coinz_Prod_Dilution";
      FP    "PulseCoinzDilutionOn";
      );
      );
      JNB   M008;
      L     0.000000e+00;
      T     "ActVolumePumps";
M008: NOP   0;
NETWORK
TITLE =
      A(;
      L     "ActVolumePumps";
      L     DB30.DBD 18;
      >=R;
      );
      AN    "Coinz_Prod_Steam_Valve";
      S     "Coinz_Prod_Steam_Valve";
      A     "cooking_end_starch";
      R     "Coinz_Prod_Steam_Valve";
      NOP   0;
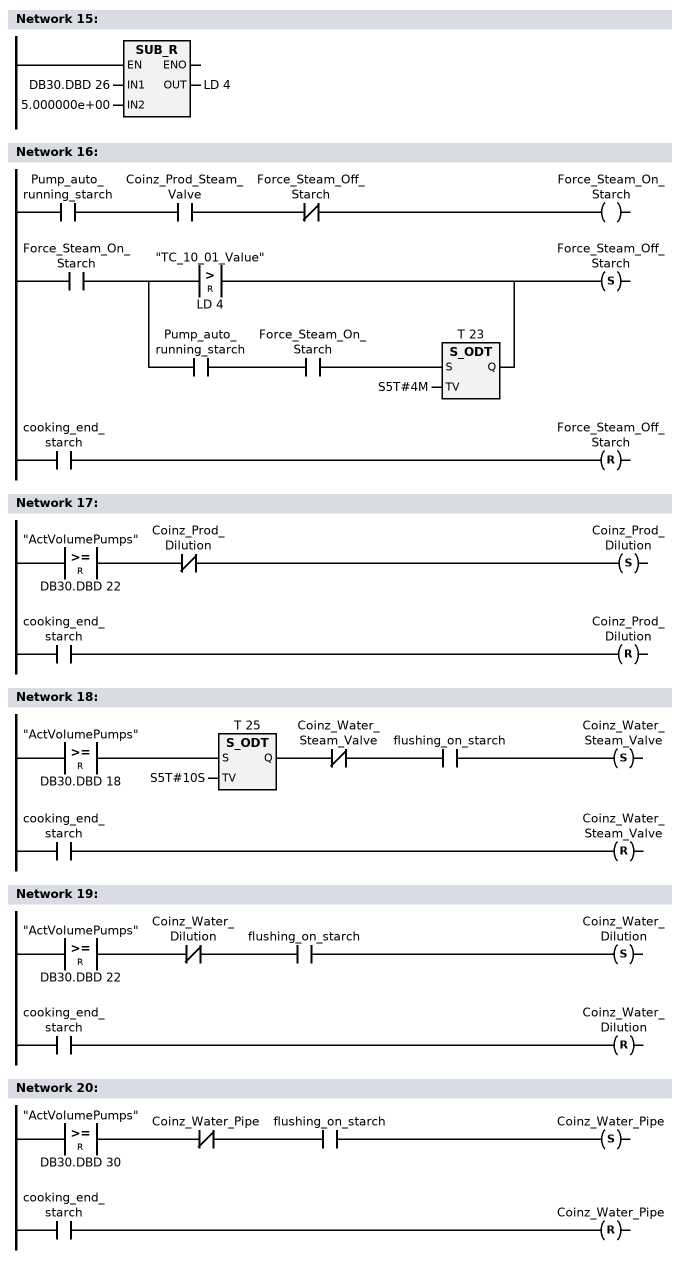
NETWORK
TITLE =
      L     DB30.DBD 26;
      L     5.000000e+00;
      -R;
      T     LD 4;
      NOP   0;
NETWORK
TITLE =
      A     "Pump_auto_running_starch";
      A     "Coinz_Prod_Steam_Valve";
      AN    "Force_Steam_Off_Starch";
      =     "Force_Steam_On_Starch";
      A     "Force_Steam_On_Starch";
      A(;
      O(;
      L     "TC_10_01_Value";
      L     LD 4;
      >R;
      );
      O(;
      A     "Pump_auto_running_starch";
      A     "Force_Steam_On_Starch";
      L     S5T#4M;
      SD    T 23;
      NOP   0;
      NOP   0;
      NOP   0;
      A     T 23;
      );
      );
      S     "Force_Steam_Off_Starch";
      A     "cooking_end_starch";
      R     "Force_Steam_Off_Starch";
      NOP   0;
NETWORK
TITLE =
      A(;
      L     "ActVolumePumps";
      L     DB30.DBD 22;
      >=R;
      );
      AN    "Coinz_Prod_Dilution";
      S     "Coinz_Prod_Dilution";
      A     "cooking_end_starch";
      R     "Coinz_Prod_Dilution";
      NOP   0;
NETWORK
TITLE =
      A(;
      A(;
      L     "ActVolumePumps";
      L     DB30.DBD 18;
      >=R;
      );
      L     S5T#10S;
      SD    T 25;
      NOP   0;
      NOP   0;
      NOP   0;
      A     T 25;
      );
      AN    "Coinz_Water_Steam_Valve";
      A     "flushing_on_starch";
      S     "Coinz_Water_Steam_Valve";
      A     "cooking_end_starch";
      R     "Coinz_Water_Steam_Valve";
      NOP   0;
NETWORK
TITLE =
      A(;
      L     "ActVolumePumps";
      L     DB30.DBD 22;
      >=R;
      );
      AN    "Coinz_Water_Dilution";
      A     "flushing_on_starch";
      S     "Coinz_Water_Dilution";
      A     "cooking_end_starch";
      R     "Coinz_Water_Dilution";
      NOP   0;
NETWORK
TITLE =
      A(;
      L     "ActVolumePumps";
      L     DB30.DBD 30;
      >=R;
      );
      AN    "Coinz_Water_Pipe";
      A     "flushing_on_starch";
      S     "Coinz_Water_Pipe";
      A     "cooking_end_starch";
      R     "Coinz_Water_Pipe";
      NOP   0;
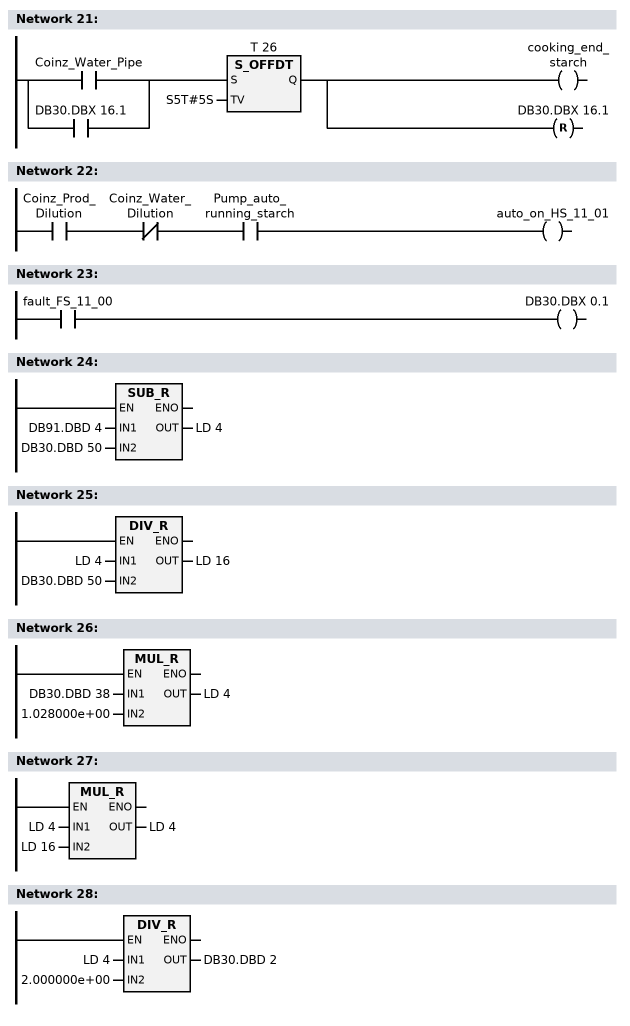
NETWORK
TITLE =
      A(;
      O     "Coinz_Water_Pipe";
      O     DB30.DBX 16.1;
      );
      L     S5T#5S;
      SF    T 26;
      NOP   0;
      NOP   0;
      NOP   0;
      A     T 26;
      =     "cooking_end_starch";
      R     DB30.DBX 16.1;
NETWORK
TITLE =
      A     "Coinz_Prod_Dilution";
      AN    "Coinz_Water_Dilution";
      A     "Pump_auto_running_starch";
      =     "auto_on_HS_11_01";
NETWORK
TITLE =
      A     "fault_FS_11_00";
      =     DB30.DBX 0.1;
NETWORK
TITLE =
      L     DB91.DBD 4;
      L     DB30.DBD 50;
      -R;
      T     LD 4;
      NOP   0;
NETWORK
TITLE =
      L     LD 4;
      L     DB30.DBD 50;
      /R;
      T     LD 16;
      NOP   0;
NETWORK
TITLE =
      L     DB30.DBD 38;
      L     1.028000e+00;
      *R;
      T     LD 4;
      NOP   0;
NETWORK
TITLE =
      L     LD 4;
      L     LD 16;
      *R;
      T     LD 4;
      NOP   0;
NETWORK
TITLE =
      L     LD 4;
      L     2.000000e+00;
      /R;
      T     DB30.DBD 2;
      NOP   0;
END_FUNCTION_BLOCK

FUNCTION_BLOCK "preparation CaCO3"	// FB 15
VERSION : 0.1
BEGIN
// (block stored without names or comments; labels and parameter names are numbered)
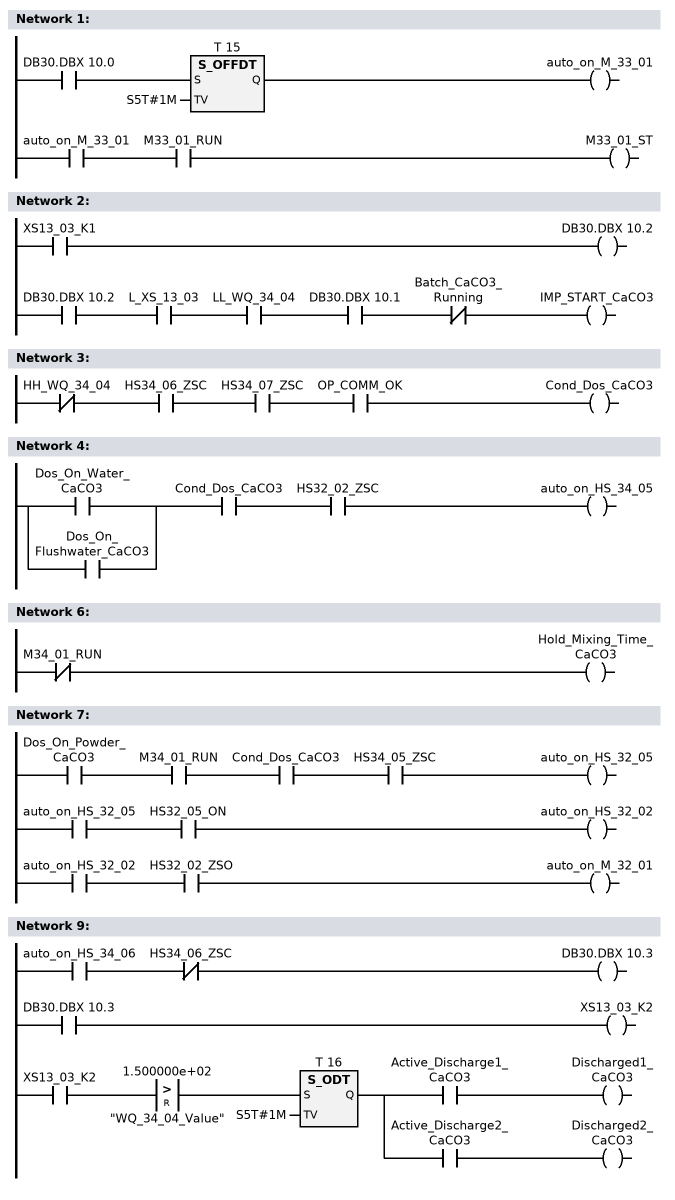
NETWORK
TITLE =
      A(;
      A     DB30.DBX 10.0;
      L     S5T#1M;
      SF    T 15;
      NOP   0;
      NOP   0;
      NOP   0;
      A     T 15;
      );
      =     "auto_on_M_33_01";
      A     "auto_on_M_33_01";
      A     "M33_01_RUN";
      =     "M33_01_ST";
NETWORK
TITLE =
      A     "XS13_03_K1";
      =     DB30.DBX 10.2;
      A     DB30.DBX 10.2;
      A     "L_XS_13_03";
      A     "LL_WQ_34_04";
      A     DB30.DBX 10.1;
      AN    "Batch_CaCO3_Running";
      =     "IMP_START_CaCO3";
NETWORK
TITLE =
      AN    "HH_WQ_34_04";
      A     "HS34_06_ZSC";
      A     "HS34_07_ZSC";
      A     "OP_COMM_OK";
      =     "Cond_Dos_CaCO3";
NETWORK
TITLE =
      A(;
      O     "Dos_On_Water_CaCO3";
      O     "Dos_On_Flushwater_CaCO3";
      );
      A     "Cond_Dos_CaCO3";
      A     "HS32_02_ZSC";
      =     "auto_on_HS_34_05";
NETWORK
TITLE =
      AN    "LL_WQ_34_04";
      A     "Cmd_Agitator_On_CaCO3";
      A(;
      A(;
      A     "Cmd_Discharge1_On_CaCO3";
      A     "L_WQ_34_04";
      S     "Agitator_Stop_CaCO3";
      AN    "Batch_CaCO3_Running";
      R     "Agitator_Stop_CaCO3";
      A     "Agitator_Stop_CaCO3";
      );
      NOT;
      );
      =     "auto_on_M_34_01";
NETWORK
TITLE =
      AN    "M34_01_RUN";
      =     "Hold_Mixing_Time_CaCO3";
NETWORK
TITLE =
      A     "Dos_On_Powder_CaCO3";
      A     "M34_01_RUN";
      A     "Cond_Dos_CaCO3";
      A     "HS34_05_ZSC";
      =     "auto_on_HS_32_05";
      A     "auto_on_HS_32_05";
      A     "HS32_05_ON";
      =     "auto_on_HS_32_02";
      A     "auto_on_HS_32_02";
      A     "HS32_02_ZSO";
      =     "auto_on_M_32_01";
NETWORK
TITLE =
      A(;
      A(;
      A     "XS13_03_K1";
      A     "L_XS_13_03";
      O(;
      A     "auto_on_HS_34_06";
      A     "Active_Discharge1_CaCO3";
      S     "Save_Dis_On_CaCO3";
      AN    "Active_Discharge1_CaCO3";
      R     "Save_Dis_On_CaCO3";
      A     "Save_Dis_On_CaCO3";
      );
      );
      A     "Cmd_Discharge1_On_CaCO3";
      A     "Active_Discharge1_CaCO3";
      O;
      A     "Cmd_Discharge2_On_CaCO3";
      A     "Active_Discharge2_CaCO3";
      );
      AN    "HH_XS_13_03";
      =     "auto_on_HS_34_06";
NETWORK
TITLE =
      A     "auto_on_HS_34_06";
      AN    "HS34_06_ZSC";
      =     DB30.DBX 10.3;
      A     DB30.DBX 10.3;
      =     "XS13_03_K2";
      A     "XS13_03_K2";
      A(;
      L     1.500000e+02;
      L     "WQ_34_04_Value";
      >R;
      );
      L     S5T#1M;
      SD    T 16;
      NOP   0;
      NOP   0;
      NOP   0;
      A     T 16;
      =     L 0.0;
      A     L 0.0;
      A     "Active_Discharge1_CaCO3";
      =     "Discharged1_CaCO3";
      A     L 0.0;
      A     "Active_Discharge2_CaCO3";
      =     "Discharged2_CaCO3";
END_FUNCTION_BLOCK

FUNCTION_BLOCK "Devices"	// FB 20
VERSION : 0.1
VAR_TEMP
  TEMP0 : INT ;
  TEMP1 : REAL ;
  TEMP2 : REAL ;
  TEMP3 : REAL ;
  TEMP4 : REAL ;
  TEMP5 : REAL ;
  TEMP6 : REAL ;
  TEMP7 : REAL ;
  TEMP8 : REAL ;
  TEMP9 : REAL ;
  TEMP10 : BOOL ;
  TEMP11 : REAL ;
  TEMP12 : REAL ;
  TEMP13 : REAL ;
  TEMP14 : REAL ;
END_VAR
BEGIN
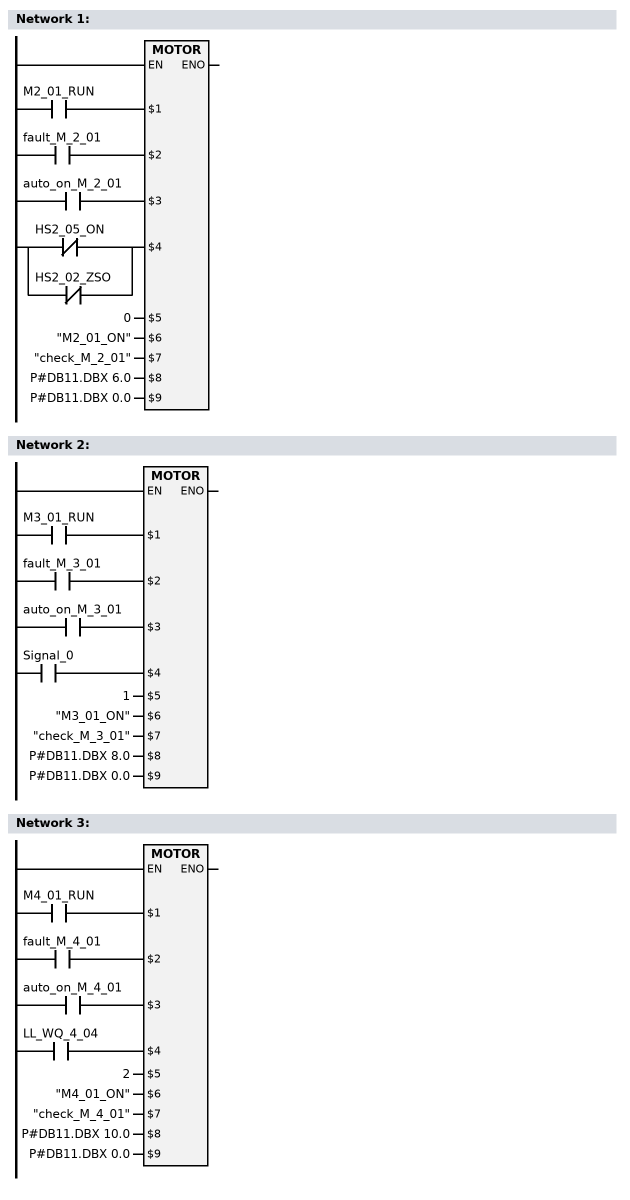
NETWORK
TITLE =
      A     "M2_01_RUN";
      =     L 56.0;
      BLD   103;
      A     "fault_M_2_01";
      =     L 56.1;
      BLD   103;
      A     "auto_on_M_2_01";
      =     L 56.2;
      BLD   103;
      A(;
      ON    "HS2_05_ON";
      ON    "HS2_02_ZSO";
      );
      =     L 56.3;
      BLD   103;
      CALL  "MOTOR" (
           $1                       := L 56.0,
           $2                       := L 56.1,
           $3                       := L 56.2,
           $4                       := L 56.3,
           $5                       := 0,
           $6                       := "M2_01_ON",
           $7                       := "check_M_2_01",
           $8                       := P#DB11.DBX 6.0,
           $9                       := P#DB11.DBX 0.0);
      NOP   0;
NETWORK
TITLE =
      A     "M3_01_RUN";
      =     L 56.0;
      BLD   103;
      A     "fault_M_3_01";
      =     L 56.1;
      BLD   103;
      A     "auto_on_M_3_01";
      =     L 56.2;
      BLD   103;
      A     "Signal_0";
      =     L 56.3;
      BLD   103;
      CALL  "MOTOR" (
           $1                       := L 56.0,
           $2                       := L 56.1,
           $3                       := L 56.2,
           $4                       := L 56.3,
           $5                       := 1,
           $6                       := "M3_01_ON",
           $7                       := "check_M_3_01",
           $8                       := P#DB11.DBX 8.0,
           $9                       := P#DB11.DBX 0.0);
      NOP   0;
NETWORK
TITLE =
      A     "M4_01_RUN";
      =     L 56.0;
      BLD   103;
      A     "fault_M_4_01";
      =     L 56.1;
      BLD   103;
      A     "auto_on_M_4_01";
      =     L 56.2;
      BLD   103;
      A     "LL_WQ_4_04";
      =     L 56.3;
      BLD   103;
      CALL  "MOTOR" (
           $1                       := L 56.0,
           $2                       := L 56.1,
           $3                       := L 56.2,
           $4                       := L 56.3,
           $5                       := 2,
           $6                       := "M4_01_ON",
           $7                       := "check_M_4_01",
           $8                       := P#DB11.DBX 10.0,
           $9                       := P#DB11.DBX 0.0);
      NOP   0;
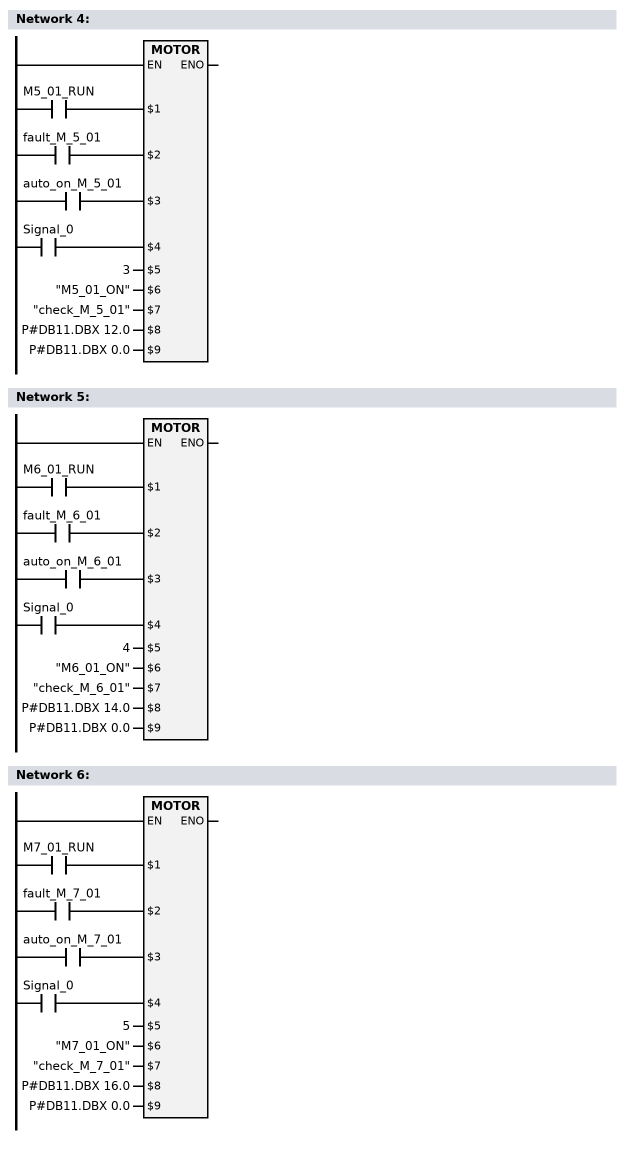
NETWORK
TITLE =
      A     "M5_01_RUN";
      =     L 56.0;
      BLD   103;
      A     "fault_M_5_01";
      =     L 56.1;
      BLD   103;
      A     "auto_on_M_5_01";
      =     L 56.2;
      BLD   103;
      A     "Signal_0";
      =     L 56.3;
      BLD   103;
      CALL  "MOTOR" (
           $1                       := L 56.0,
           $2                       := L 56.1,
           $3                       := L 56.2,
           $4                       := L 56.3,
           $5                       := 3,
           $6                       := "M5_01_ON",
           $7                       := "check_M_5_01",
           $8                       := P#DB11.DBX 12.0,
           $9                       := P#DB11.DBX 0.0);
      NOP   0;
NETWORK
TITLE =
      A     "M6_01_RUN";
      =     L 56.0;
      BLD   103;
      A     "fault_M_6_01";
      =     L 56.1;
      BLD   103;
      A     "auto_on_M_6_01";
      =     L 56.2;
      BLD   103;
      A     "Signal_0";
      =     L 56.3;
      BLD   103;
      CALL  "MOTOR" (
           $1                       := L 56.0,
           $2                       := L 56.1,
           $3                       := L 56.2,
           $4                       := L 56.3,
           $5                       := 4,
           $6                       := "M6_01_ON",
           $7                       := "check_M_6_01",
           $8                       := P#DB11.DBX 14.0,
           $9                       := P#DB11.DBX 0.0);
      NOP   0;
NETWORK
TITLE =
      A     "M7_01_RUN";
      =     L 56.0;
      BLD   103;
      A     "fault_M_7_01";
      =     L 56.1;
      BLD   103;
      A     "auto_on_M_7_01";
      =     L 56.2;
      BLD   103;
      A     "Signal_0";
      =     L 56.3;
      BLD   103;
      CALL  "MOTOR" (
           $1                       := L 56.0,
           $2                       := L 56.1,
           $3                       := L 56.2,
           $4                       := L 56.3,
           $5                       := 5,
           $6                       := "M7_01_ON",
           $7                       := "check_M_7_01",
           $8                       := P#DB11.DBX 16.0,
           $9                       := P#DB11.DBX 0.0);
      NOP   0;
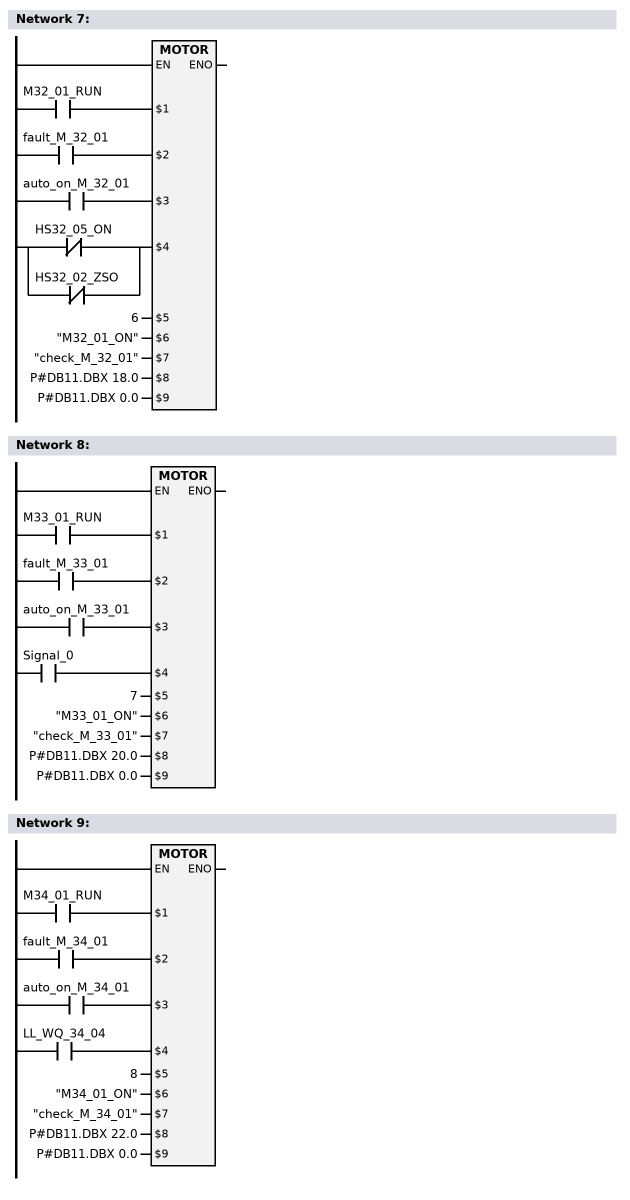
NETWORK
TITLE =
      A     "M32_01_RUN";
      =     L 56.0;
      BLD   103;
      A     "fault_M_32_01";
      =     L 56.1;
      BLD   103;
      A     "auto_on_M_32_01";
      =     L 56.2;
      BLD   103;
      A(;
      ON    "HS32_05_ON";
      ON    "HS32_02_ZSO";
      );
      =     L 56.3;
      BLD   103;
      CALL  "MOTOR" (
           $1                       := L 56.0,
           $2                       := L 56.1,
           $3                       := L 56.2,
           $4                       := L 56.3,
           $5                       := 6,
           $6                       := "M32_01_ON",
           $7                       := "check_M_32_01",
           $8                       := P#DB11.DBX 18.0,
           $9                       := P#DB11.DBX 0.0);
      NOP   0;
NETWORK
TITLE =
      A     "M33_01_RUN";
      =     L 56.0;
      BLD   103;
      A     "fault_M_33_01";
      =     L 56.1;
      BLD   103;
      A     "auto_on_M_33_01";
      =     L 56.2;
      BLD   103;
      A     "Signal_0";
      =     L 56.3;
      BLD   103;
      CALL  "MOTOR" (
           $1                       := L 56.0,
           $2                       := L 56.1,
           $3                       := L 56.2,
           $4                       := L 56.3,
           $5                       := 7,
           $6                       := "M33_01_ON",
           $7                       := "check_M_33_01",
           $8                       := P#DB11.DBX 20.0,
           $9                       := P#DB11.DBX 0.0);
      NOP   0;
NETWORK
TITLE =
      A     "M34_01_RUN";
      =     L 56.0;
      BLD   103;
      A     "fault_M_34_01";
      =     L 56.1;
      BLD   103;
      A     "auto_on_M_34_01";
      =     L 56.2;
      BLD   103;
      A     "LL_WQ_34_04";
      =     L 56.3;
      BLD   103;
      CALL  "MOTOR" (
           $1                       := L 56.0,
           $2                       := L 56.1,
           $3                       := L 56.2,
           $4                       := L 56.3,
           $5                       := 8,
           $6                       := "M34_01_ON",
           $7                       := "check_M_34_01",
           $8                       := P#DB11.DBX 22.0,
           $9                       := P#DB11.DBX 0.0);
      NOP   0;
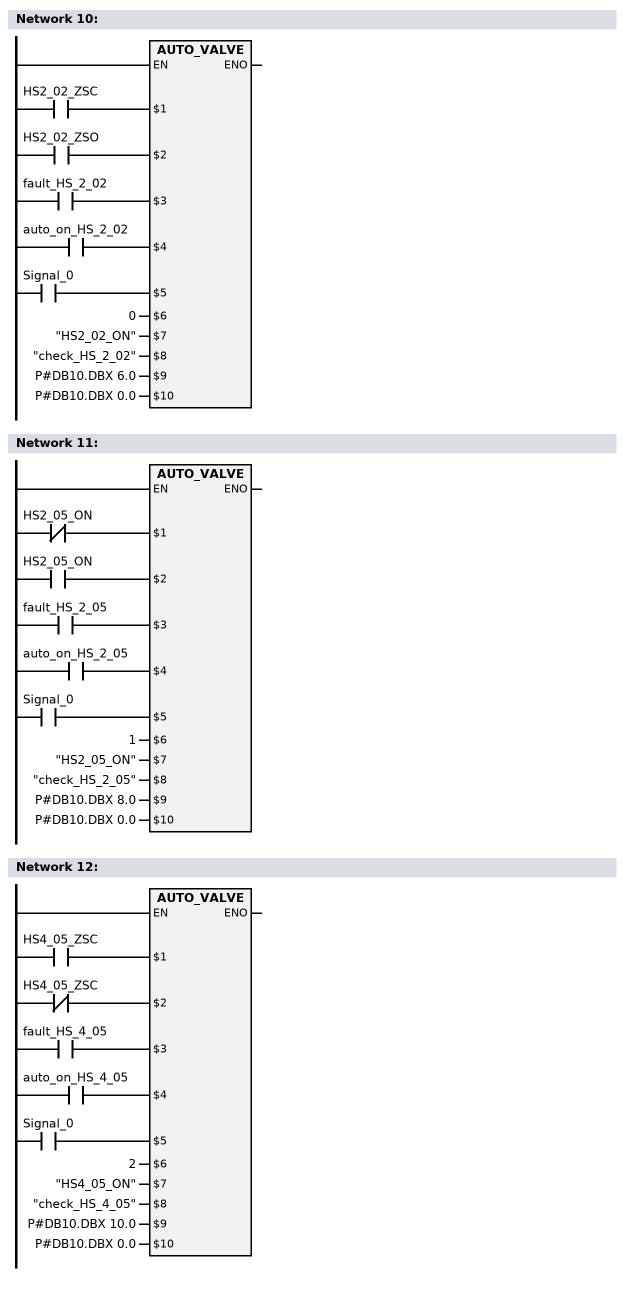
NETWORK
TITLE =
      A     "HS2_02_ZSC";
      =     L 56.0;
      BLD   103;
      A     "HS2_02_ZSO";
      =     L 56.1;
      BLD   103;
      A     "fault_HS_2_02";
      =     L 56.2;
      BLD   103;
      A     "auto_on_HS_2_02";
      =     L 56.3;
      BLD   103;
      A     "Signal_0";
      =     L 56.4;
      BLD   103;
      CALL  "AUTO_VALVE" (
           $1                       := L 56.0,
           $2                       := L 56.1,
           $3                       := L 56.2,
           $4                       := L 56.3,
           $5                       := L 56.4,
           $6                       := 0,
           $7                       := "HS2_02_ON",
           $8                       := "check_HS_2_02",
           $9                       := P#DB10.DBX 6.0,
           $10                      := P#DB10.DBX 0.0);
      NOP   0;
NETWORK
TITLE =
      AN    "HS2_05_ON";
      =     L 56.0;
      BLD   103;
      A     "HS2_05_ON";
      =     L 56.1;
      BLD   103;
      A     "fault_HS_2_05";
      =     L 56.2;
      BLD   103;
      A     "auto_on_HS_2_05";
      =     L 56.3;
      BLD   103;
      A     "Signal_0";
      =     L 56.4;
      BLD   103;
      CALL  "AUTO_VALVE" (
           $1                       := L 56.0,
           $2                       := L 56.1,
           $3                       := L 56.2,
           $4                       := L 56.3,
           $5                       := L 56.4,
           $6                       := 1,
           $7                       := "HS2_05_ON",
           $8                       := "check_HS_2_05",
           $9                       := P#DB10.DBX 8.0,
           $10                      := P#DB10.DBX 0.0);
      NOP   0;
NETWORK
TITLE =
      A     "HS4_05_ZSC";
      =     L 56.0;
      BLD   103;
      AN    "HS4_05_ZSC";
      =     L 56.1;
      BLD   103;
      A     "fault_HS_4_05";
      =     L 56.2;
      BLD   103;
      A     "auto_on_HS_4_05";
      =     L 56.3;
      BLD   103;
      A     "Signal_0";
      =     L 56.4;
      BLD   103;
      CALL  "AUTO_VALVE" (
           $1                       := L 56.0,
           $2                       := L 56.1,
           $3                       := L 56.2,
           $4                       := L 56.3,
           $5                       := L 56.4,
           $6                       := 2,
           $7                       := "HS4_05_ON",
           $8                       := "check_HS_4_05",
           $9                       := P#DB10.DBX 10.0,
           $10                      := P#DB10.DBX 0.0);
      NOP   0;
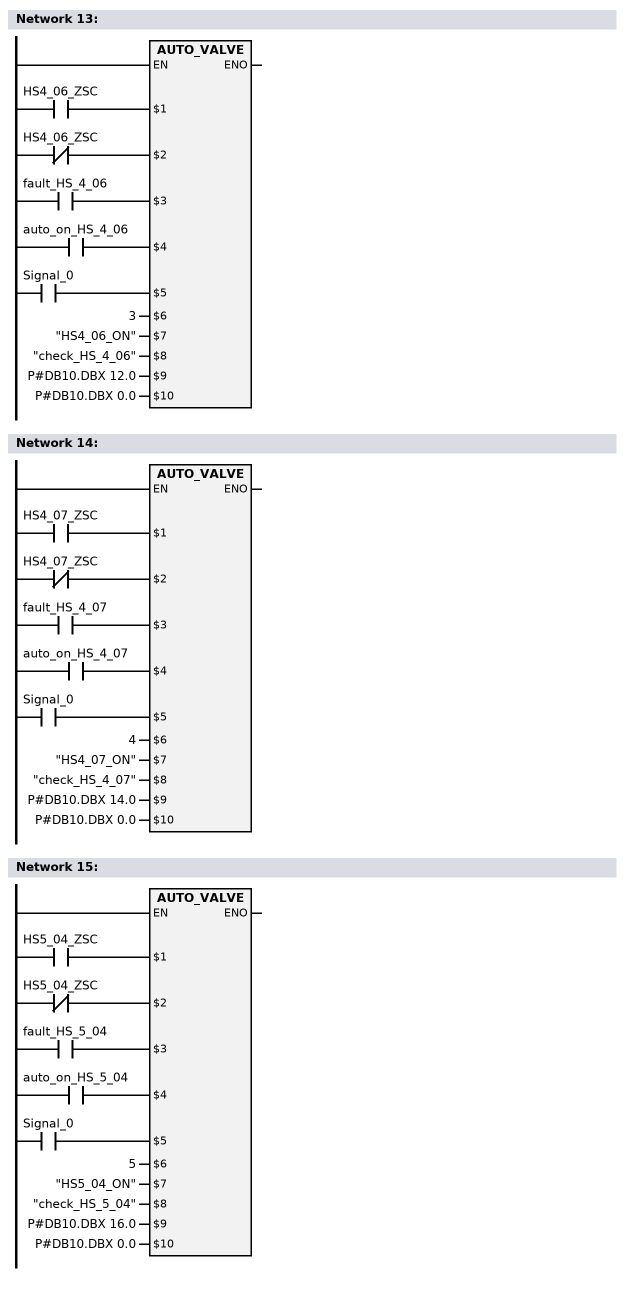
NETWORK
TITLE =
      A     "HS4_06_ZSC";
      =     L 56.0;
      BLD   103;
      AN    "HS4_06_ZSC";
      =     L 56.1;
      BLD   103;
      A     "fault_HS_4_06";
      =     L 56.2;
      BLD   103;
      A     "auto_on_HS_4_06";
      =     L 56.3;
      BLD   103;
      A     "Signal_0";
      =     L 56.4;
      BLD   103;
      CALL  "AUTO_VALVE" (
           $1                       := L 56.0,
           $2                       := L 56.1,
           $3                       := L 56.2,
           $4                       := L 56.3,
           $5                       := L 56.4,
           $6                       := 3,
           $7                       := "HS4_06_ON",
           $8                       := "check_HS_4_06",
           $9                       := P#DB10.DBX 12.0,
           $10                      := P#DB10.DBX 0.0);
      NOP   0;
NETWORK
TITLE =
      A     "HS4_07_ZSC";
      =     L 56.0;
      BLD   103;
      AN    "HS4_07_ZSC";
      =     L 56.1;
      BLD   103;
      A     "fault_HS_4_07";
      =     L 56.2;
      BLD   103;
      A     "auto_on_HS_4_07";
      =     L 56.3;
      BLD   103;
      A     "Signal_0";
      =     L 56.4;
      BLD   103;
      CALL  "AUTO_VALVE" (
           $1                       := L 56.0,
           $2                       := L 56.1,
           $3                       := L 56.2,
           $4                       := L 56.3,
           $5                       := L 56.4,
           $6                       := 4,
           $7                       := "HS4_07_ON",
           $8                       := "check_HS_4_07",
           $9                       := P#DB10.DBX 14.0,
           $10                      := P#DB10.DBX 0.0);
      NOP   0;
NETWORK
TITLE =
      A     "HS5_04_ZSC";
      =     L 56.0;
      BLD   103;
      AN    "HS5_04_ZSC";
      =     L 56.1;
      BLD   103;
      A     "fault_HS_5_04";
      =     L 56.2;
      BLD   103;
      A     "auto_on_HS_5_04";
      =     L 56.3;
      BLD   103;
      A     "Signal_0";
      =     L 56.4;
      BLD   103;
      CALL  "AUTO_VALVE" (
           $1                       := L 56.0,
           $2                       := L 56.1,
           $3                       := L 56.2,
           $4                       := L 56.3,
           $5                       := L 56.4,
           $6                       := 5,
           $7                       := "HS5_04_ON",
           $8                       := "check_HS_5_04",
           $9                       := P#DB10.DBX 16.0,
           $10                      := P#DB10.DBX 0.0);
      NOP   0;
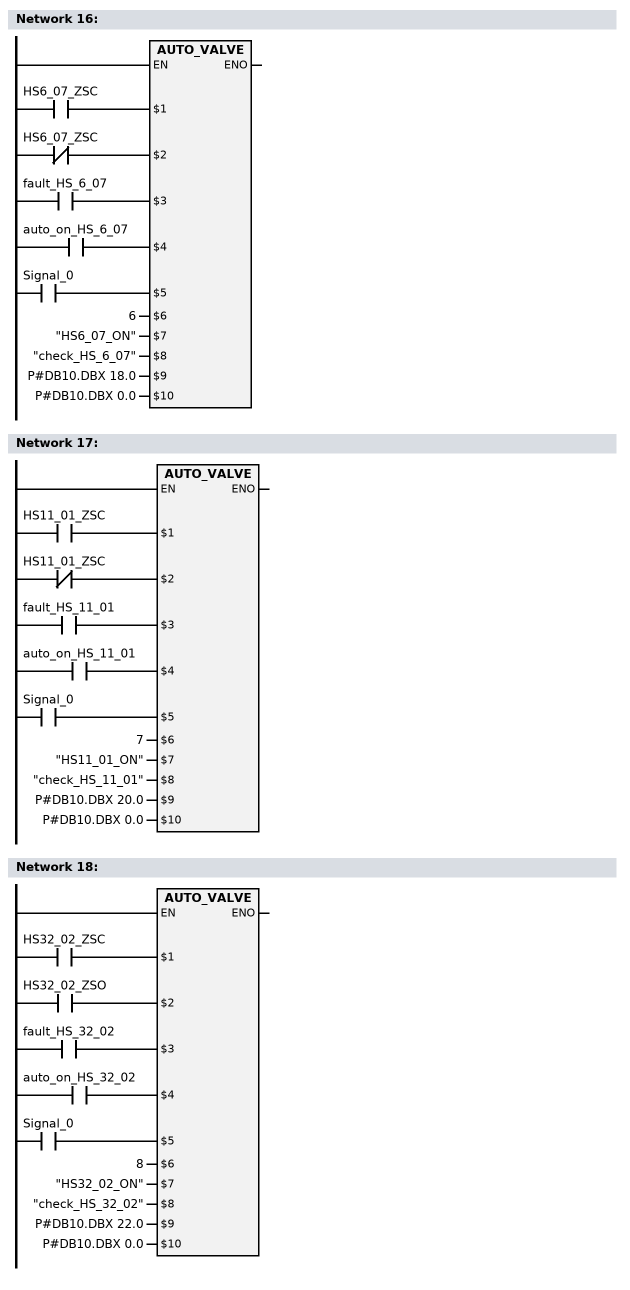
NETWORK
TITLE =
      A     "HS6_07_ZSC";
      =     L 56.0;
      BLD   103;
      AN    "HS6_07_ZSC";
      =     L 56.1;
      BLD   103;
      A     "fault_HS_6_07";
      =     L 56.2;
      BLD   103;
      A     "auto_on_HS_6_07";
      =     L 56.3;
      BLD   103;
      A     "Signal_0";
      =     L 56.4;
      BLD   103;
      CALL  "AUTO_VALVE" (
           $1                       := L 56.0,
           $2                       := L 56.1,
           $3                       := L 56.2,
           $4                       := L 56.3,
           $5                       := L 56.4,
           $6                       := 6,
           $7                       := "HS6_07_ON",
           $8                       := "check_HS_6_07",
           $9                       := P#DB10.DBX 18.0,
           $10                      := P#DB10.DBX 0.0);
      NOP   0;
NETWORK
TITLE =
      A     "HS11_01_ZSC";
      =     L 56.0;
      BLD   103;
      AN    "HS11_01_ZSC";
      =     L 56.1;
      BLD   103;
      A     "fault_HS_11_01";
      =     L 56.2;
      BLD   103;
      A     "auto_on_HS_11_01";
      =     L 56.3;
      BLD   103;
      A     "Signal_0";
      =     L 56.4;
      BLD   103;
      CALL  "AUTO_VALVE" (
           $1                       := L 56.0,
           $2                       := L 56.1,
           $3                       := L 56.2,
           $4                       := L 56.3,
           $5                       := L 56.4,
           $6                       := 7,
           $7                       := "HS11_01_ON",
           $8                       := "check_HS_11_01",
           $9                       := P#DB10.DBX 20.0,
           $10                      := P#DB10.DBX 0.0);
      NOP   0;
NETWORK
TITLE =
      A     "HS32_02_ZSC";
      =     L 56.0;
      BLD   103;
      A     "HS32_02_ZSO";
      =     L 56.1;
      BLD   103;
      A     "fault_HS_32_02";
      =     L 56.2;
      BLD   103;
      A     "auto_on_HS_32_02";
      =     L 56.3;
      BLD   103;
      A     "Signal_0";
      =     L 56.4;
      BLD   103;
      CALL  "AUTO_VALVE" (
           $1                       := L 56.0,
           $2                       := L 56.1,
           $3                       := L 56.2,
           $4                       := L 56.3,
           $5                       := L 56.4,
           $6                       := 8,
           $7                       := "HS32_02_ON",
           $8                       := "check_HS_32_02",
           $9                       := P#DB10.DBX 22.0,
           $10                      := P#DB10.DBX 0.0);
      NOP   0;
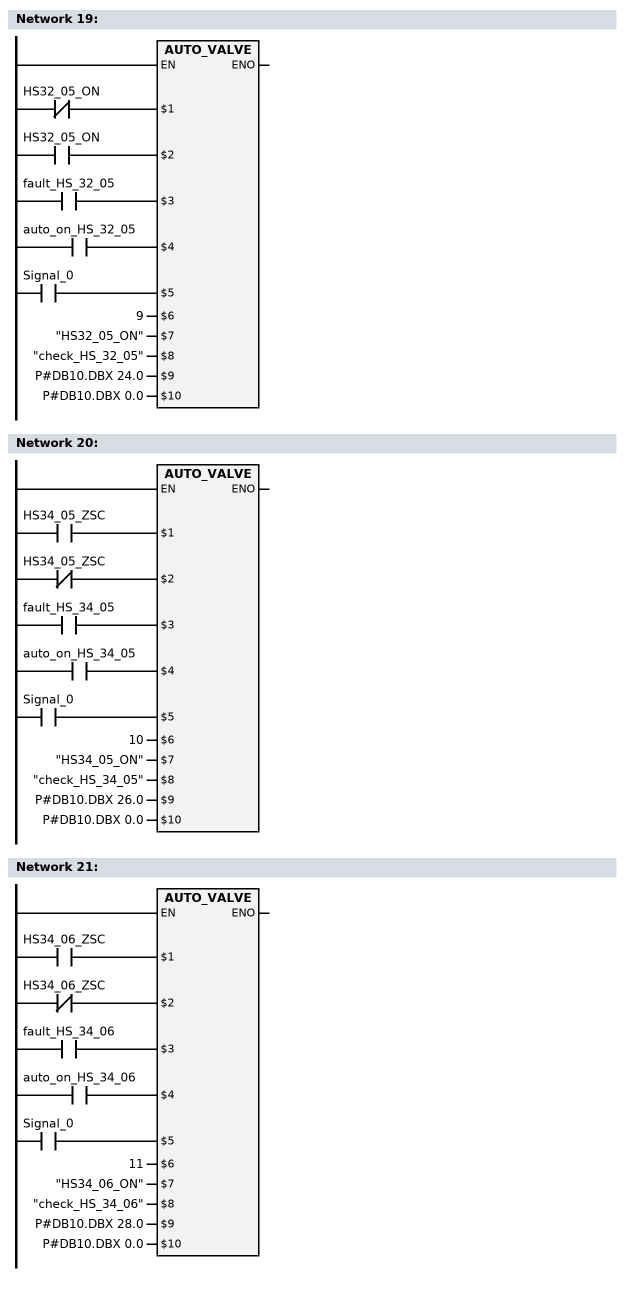
NETWORK
TITLE =
      AN    "HS32_05_ON";
      =     L 56.0;
      BLD   103;
      A     "HS32_05_ON";
      =     L 56.1;
      BLD   103;
      A     "fault_HS_32_05";
      =     L 56.2;
      BLD   103;
      A     "auto_on_HS_32_05";
      =     L 56.3;
      BLD   103;
      A     "Signal_0";
      =     L 56.4;
      BLD   103;
      CALL  "AUTO_VALVE" (
           $1                       := L 56.0,
           $2                       := L 56.1,
           $3                       := L 56.2,
           $4                       := L 56.3,
           $5                       := L 56.4,
           $6                       := 9,
           $7                       := "HS32_05_ON",
           $8                       := "check_HS_32_05",
           $9                       := P#DB10.DBX 24.0,
           $10                      := P#DB10.DBX 0.0);
      NOP   0;
NETWORK
TITLE =
      A     "HS34_05_ZSC";
      =     L 56.0;
      BLD   103;
      AN    "HS34_05_ZSC";
      =     L 56.1;
      BLD   103;
      A     "fault_HS_34_05";
      =     L 56.2;
      BLD   103;
      A     "auto_on_HS_34_05";
      =     L 56.3;
      BLD   103;
      A     "Signal_0";
      =     L 56.4;
      BLD   103;
      CALL  "AUTO_VALVE" (
           $1                       := L 56.0,
           $2                       := L 56.1,
           $3                       := L 56.2,
           $4                       := L 56.3,
           $5                       := L 56.4,
           $6                       := 10,
           $7                       := "HS34_05_ON",
           $8                       := "check_HS_34_05",
           $9                       := P#DB10.DBX 26.0,
           $10                      := P#DB10.DBX 0.0);
      NOP   0;
NETWORK
TITLE =
      A     "HS34_06_ZSC";
      =     L 56.0;
      BLD   103;
      AN    "HS34_06_ZSC";
      =     L 56.1;
      BLD   103;
      A     "fault_HS_34_06";
      =     L 56.2;
      BLD   103;
      A     "auto_on_HS_34_06";
      =     L 56.3;
      BLD   103;
      A     "Signal_0";
      =     L 56.4;
      BLD   103;
      CALL  "AUTO_VALVE" (
           $1                       := L 56.0,
           $2                       := L 56.1,
           $3                       := L 56.2,
           $4                       := L 56.3,
           $5                       := L 56.4,
           $6                       := 11,
           $7                       := "HS34_06_ON",
           $8                       := "check_HS_34_06",
           $9                       := P#DB10.DBX 28.0,
           $10                      := P#DB10.DBX 0.0);
      NOP   0;
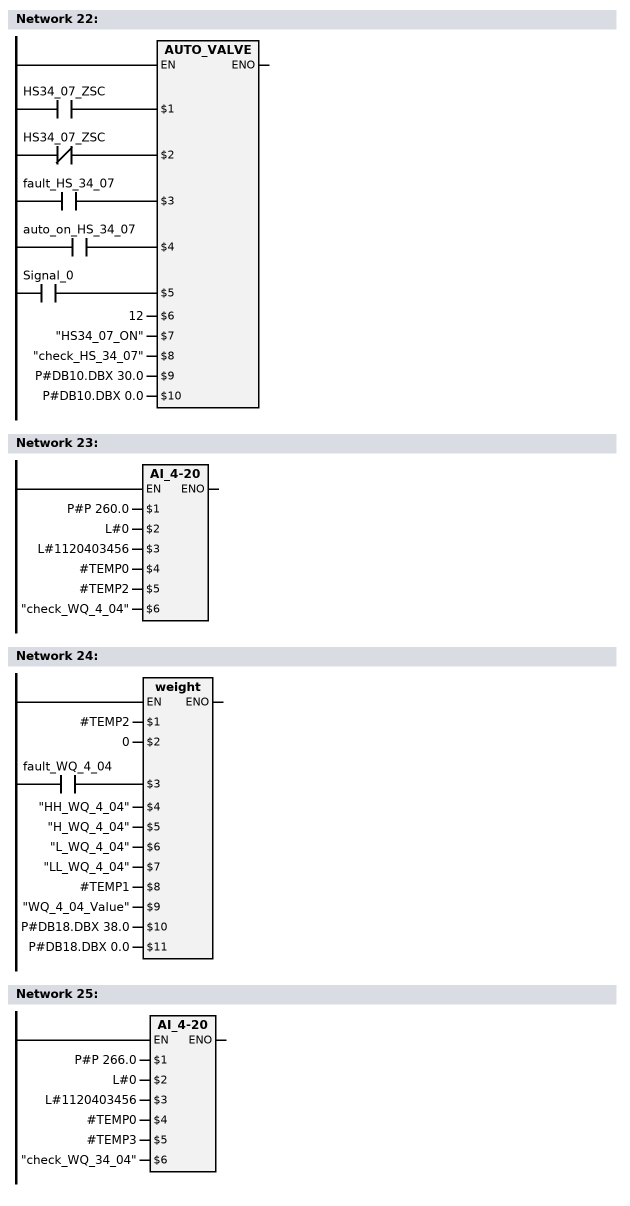
NETWORK
TITLE =
      A     "HS34_07_ZSC";
      =     L 56.0;
      BLD   103;
      AN    "HS34_07_ZSC";
      =     L 56.1;
      BLD   103;
      A     "fault_HS_34_07";
      =     L 56.2;
      BLD   103;
      A     "auto_on_HS_34_07";
      =     L 56.3;
      BLD   103;
      A     "Signal_0";
      =     L 56.4;
      BLD   103;
      CALL  "AUTO_VALVE" (
           $1                       := L 56.0,
           $2                       := L 56.1,
           $3                       := L 56.2,
           $4                       := L 56.3,
           $5                       := L 56.4,
           $6                       := 12,
           $7                       := "HS34_07_ON",
           $8                       := "check_HS_34_07",
           $9                       := P#DB10.DBX 30.0,
           $10                      := P#DB10.DBX 0.0);
      NOP   0;
NETWORK
TITLE =
      CALL  "AI_4-20" (
           $1                       := P#P 260.0,
           $2                       := L#0,
           $3                       := L#1120403456,
           $4                       := #TEMP0,
           $5                       := #TEMP2,
           $6                       := "check_WQ_4_04");
      NOP   0;
NETWORK
TITLE =
      A     "fault_WQ_4_04";
      =     L 56.0;
      BLD   103;
      CALL  "weight" (
           $1                       := #TEMP2,
           $2                       := 0,
           $3                       := L 56.0,
           $4                       := "HH_WQ_4_04",
           $5                       := "H_WQ_4_04",
           $6                       := "L_WQ_4_04",
           $7                       := "LL_WQ_4_04",
           $8                       := #TEMP1,
           $9                       := "WQ_4_04_Value",
           $10                      := P#DB18.DBX 38.0,
           $11                      := P#DB18.DBX 0.0);
      NOP   0;
NETWORK
TITLE =
      CALL  "AI_4-20" (
           $1                       := P#P 266.0,
           $2                       := L#0,
           $3                       := L#1120403456,
           $4                       := #TEMP0,
           $5                       := #TEMP3,
           $6                       := "check_WQ_34_04");
      NOP   0;
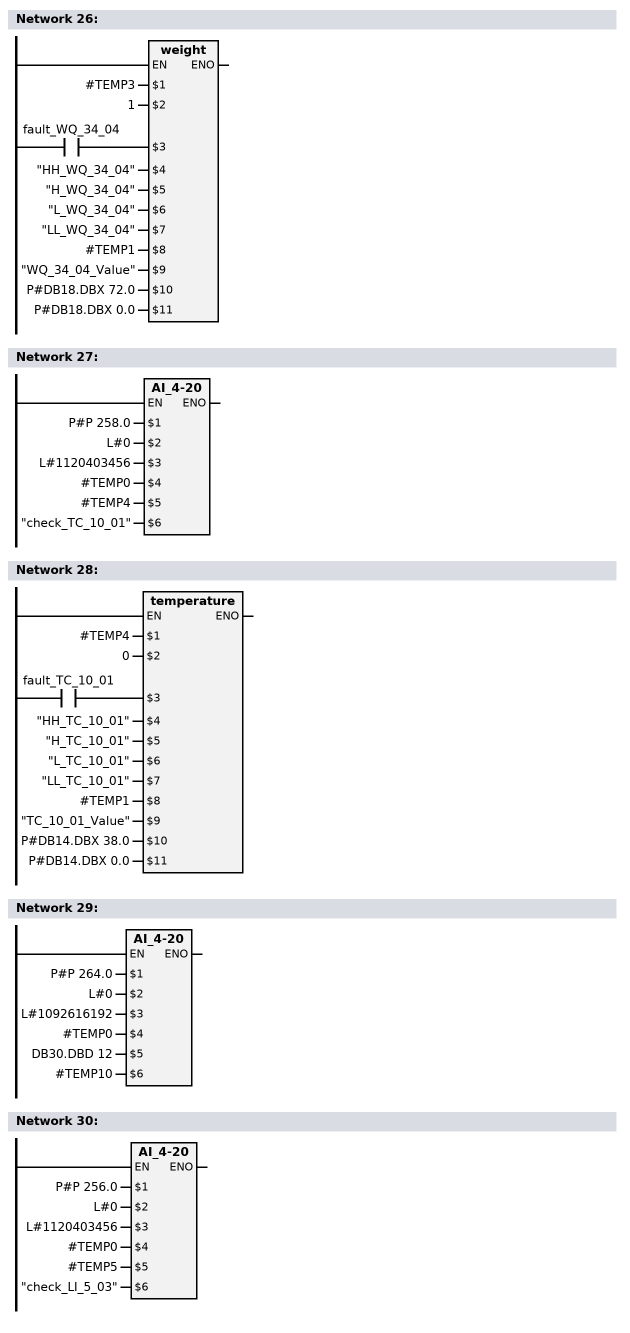
NETWORK
TITLE =
      A     "fault_WQ_34_04";
      =     L 56.0;
      BLD   103;
      CALL  "weight" (
           $1                       := #TEMP3,
           $2                       := 1,
           $3                       := L 56.0,
           $4                       := "HH_WQ_34_04",
           $5                       := "H_WQ_34_04",
           $6                       := "L_WQ_34_04",
           $7                       := "LL_WQ_34_04",
           $8                       := #TEMP1,
           $9                       := "WQ_34_04_Value",
           $10                      := P#DB18.DBX 72.0,
           $11                      := P#DB18.DBX 0.0);
      NOP   0;
NETWORK
TITLE =
      CALL  "AI_4-20" (
           $1                       := P#P 258.0,
           $2                       := L#0,
           $3                       := L#1120403456,
           $4                       := #TEMP0,
           $5                       := #TEMP4,
           $6                       := "check_TC_10_01");
      NOP   0;
NETWORK
TITLE =
      A     "fault_TC_10_01";
      =     L 56.0;
      BLD   103;
      CALL  "temperature" (
           $1                       := #TEMP4,
           $2                       := 0,
           $3                       := L 56.0,
           $4                       := "HH_TC_10_01",
           $5                       := "H_TC_10_01",
           $6                       := "L_TC_10_01",
           $7                       := "LL_TC_10_01",
           $8                       := #TEMP1,
           $9                       := "TC_10_01_Value",
           $10                      := P#DB14.DBX 38.0,
           $11                      := P#DB14.DBX 0.0);
      NOP   0;
NETWORK
TITLE =
      CALL  "AI_4-20" (
           $1                       := P#P 264.0,
           $2                       := L#0,
           $3                       := L#1092616192,
           $4                       := #TEMP0,
           $5                       := DB30.DBD 12,
           $6                       := #TEMP10);
      NOP   0;
NETWORK
TITLE =
      CALL  "AI_4-20" (
           $1                       := P#P 256.0,
           $2                       := L#0,
           $3                       := L#1120403456,
           $4                       := #TEMP0,
           $5                       := #TEMP5,
           $6                       := "check_LI_5_03");
      NOP   0;
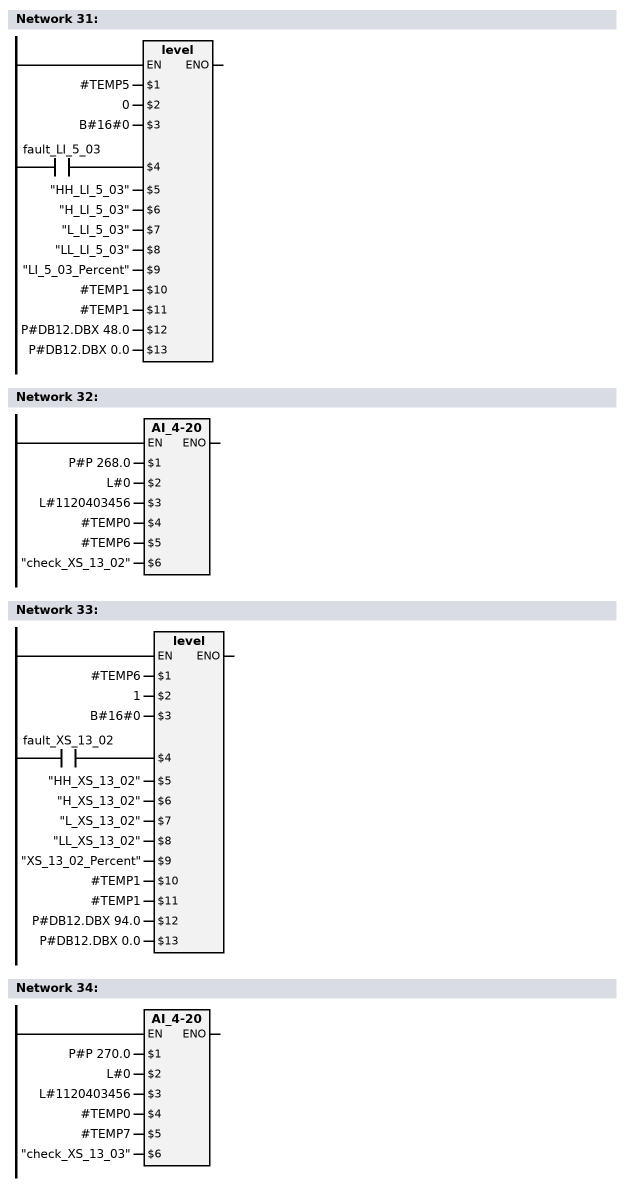
NETWORK
TITLE =
      A     "fault_LI_5_03";
      =     L 56.0;
      BLD   103;
      CALL  "level" (
           $1                       := #TEMP5,
           $2                       := 0,
           $3                       := B#16#0,
           $4                       := L 56.0,
           $5                       := "HH_LI_5_03",
           $6                       := "H_LI_5_03",
           $7                       := "L_LI_5_03",
           $8                       := "LL_LI_5_03",
           $9                       := "LI_5_03_Percent",
           $10                      := #TEMP1,
           $11                      := #TEMP1,
           $12                      := P#DB12.DBX 48.0,
           $13                      := P#DB12.DBX 0.0);
      NOP   0;
NETWORK
TITLE =
      CALL  "AI_4-20" (
           $1                       := P#P 268.0,
           $2                       := L#0,
           $3                       := L#1120403456,
           $4                       := #TEMP0,
           $5                       := #TEMP6,
           $6                       := "check_XS_13_02");
      NOP   0;
NETWORK
TITLE =
      A     "fault_XS_13_02";
      =     L 56.0;
      BLD   103;
      CALL  "level" (
           $1                       := #TEMP6,
           $2                       := 1,
           $3                       := B#16#0,
           $4                       := L 56.0,
           $5                       := "HH_XS_13_02",
           $6                       := "H_XS_13_02",
           $7                       := "L_XS_13_02",
           $8                       := "LL_XS_13_02",
           $9                       := "XS_13_02_Percent",
           $10                      := #TEMP1,
           $11                      := #TEMP1,
           $12                      := P#DB12.DBX 94.0,
           $13                      := P#DB12.DBX 0.0);
      NOP   0;
NETWORK
TITLE =
      CALL  "AI_4-20" (
           $1                       := P#P 270.0,
           $2                       := L#0,
           $3                       := L#1120403456,
           $4                       := #TEMP0,
           $5                       := #TEMP7,
           $6                       := "check_XS_13_03");
      NOP   0;
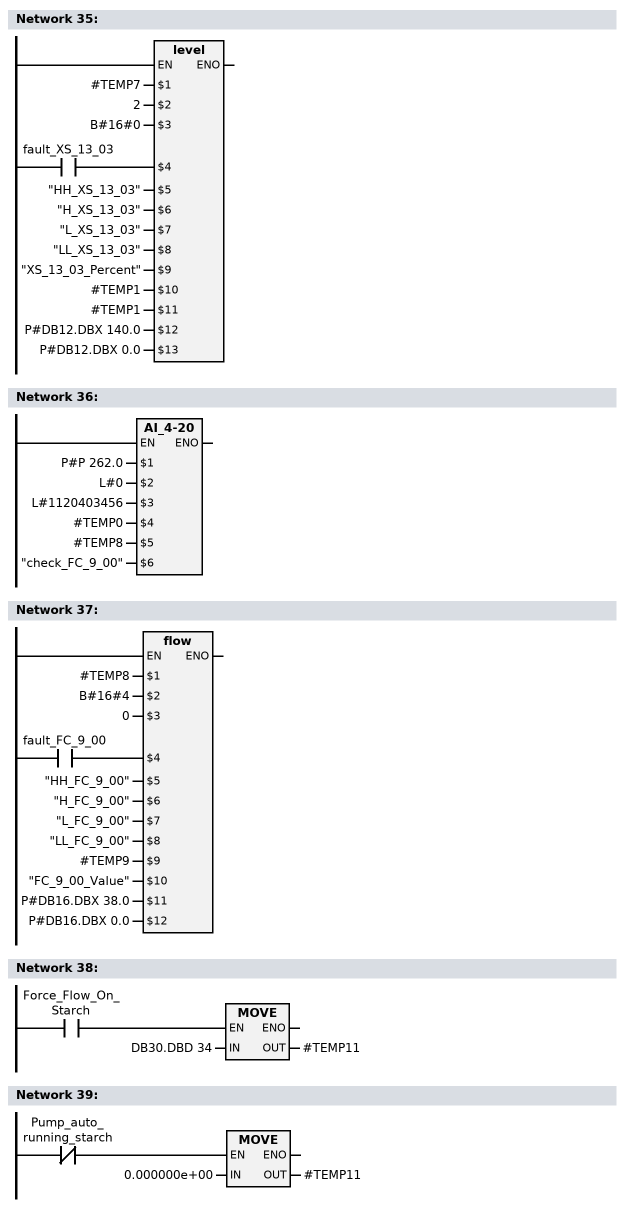
NETWORK
TITLE =
      A     "fault_XS_13_03";
      =     L 56.0;
      BLD   103;
      CALL  "level" (
           $1                       := #TEMP7,
           $2                       := 2,
           $3                       := B#16#0,
           $4                       := L 56.0,
           $5                       := "HH_XS_13_03",
           $6                       := "H_XS_13_03",
           $7                       := "L_XS_13_03",
           $8                       := "LL_XS_13_03",
           $9                       := "XS_13_03_Percent",
           $10                      := #TEMP1,
           $11                      := #TEMP1,
           $12                      := P#DB12.DBX 140.0,
           $13                      := P#DB12.DBX 0.0);
      NOP   0;
NETWORK
TITLE =
      CALL  "AI_4-20" (
           $1                       := P#P 262.0,
           $2                       := L#0,
           $3                       := L#1120403456,
           $4                       := #TEMP0,
           $5                       := #TEMP8,
           $6                       := "check_FC_9_00");
      NOP   0;
NETWORK
TITLE =
      A     "fault_FC_9_00";
      =     L 56.0;
      BLD   103;
      CALL  "flow" (
           $1                       := #TEMP8,
           $2                       := B#16#4,
           $3                       := 0,
           $4                       := L 56.0,
           $5                       := "HH_FC_9_00",
           $6                       := "H_FC_9_00",
           $7                       := "L_FC_9_00",
           $8                       := "LL_FC_9_00",
           $9                       := #TEMP9,
           $10                      := "FC_9_00_Value",
           $11                      := P#DB16.DBX 38.0,
           $12                      := P#DB16.DBX 0.0);
      NOP   0;
NETWORK
TITLE =
      A     "Force_Flow_On_Starch";
      JNB   _001;
      L     DB30.DBD 34;
      T     #TEMP11;
_001: NOP   0;
NETWORK
TITLE =
      AN    "Pump_auto_running_starch";
      JNB   _002;
      L     0.000000e+00;
      T     #TEMP11;
_002: NOP   0;
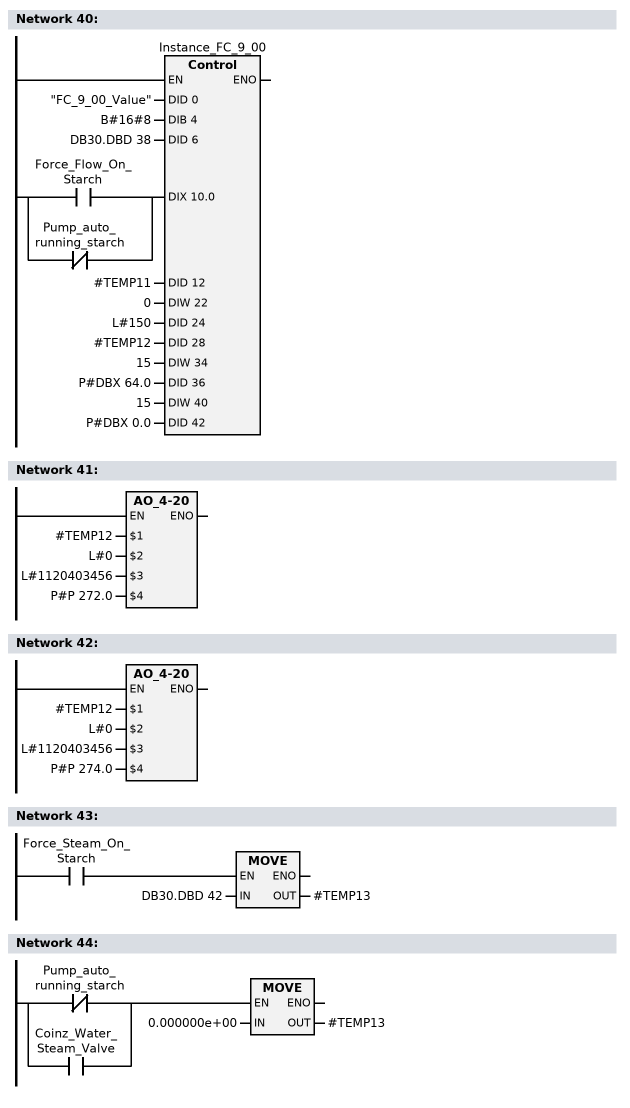
NETWORK
TITLE =
      A(;
      O     "Force_Flow_On_Starch";
      ON    "Pump_auto_running_starch";
      );
      =     L 56.0;
      BLD   103;
      CALL  "Control" , "Instance_FC_9_00" (
           DID 0                    := "FC_9_00_Value",
           DIB 4                    := B#16#8,
           DID 6                    := DB30.DBD 38,
           DIX 10.0                 := L 56.0,
           DID 12                   := #TEMP11,
           DIW 22                   := 0,
           DID 24                   := L#150,
           DID 28                   := #TEMP12,
           DIW 34                   := 15,
           DID 36                   := P#DBX 64.0,
           DIW 40                   := 15,
           DID 42                   := P#DBX 0.0);
      NOP   0;
NETWORK
TITLE =
      CALL  "AO_4-20" (
           $1                       := #TEMP12,
           $2                       := L#0,
           $3                       := L#1120403456,
           $4                       := P#P 272.0);
      NOP   0;
NETWORK
TITLE =
      CALL  "AO_4-20" (
           $1                       := #TEMP12,
           $2                       := L#0,
           $3                       := L#1120403456,
           $4                       := P#P 274.0);
      NOP   0;
NETWORK
TITLE =
      A     "Force_Steam_On_Starch";
      JNB   _003;
      L     DB30.DBD 42;
      T     #TEMP13;
_003: NOP   0;
NETWORK
TITLE =
      A(;
      ON    "Pump_auto_running_starch";
      O     "Coinz_Water_Steam_Valve";
      );
      JNB   _004;
      L     0.000000e+00;
      T     #TEMP13;
_004: NOP   0;
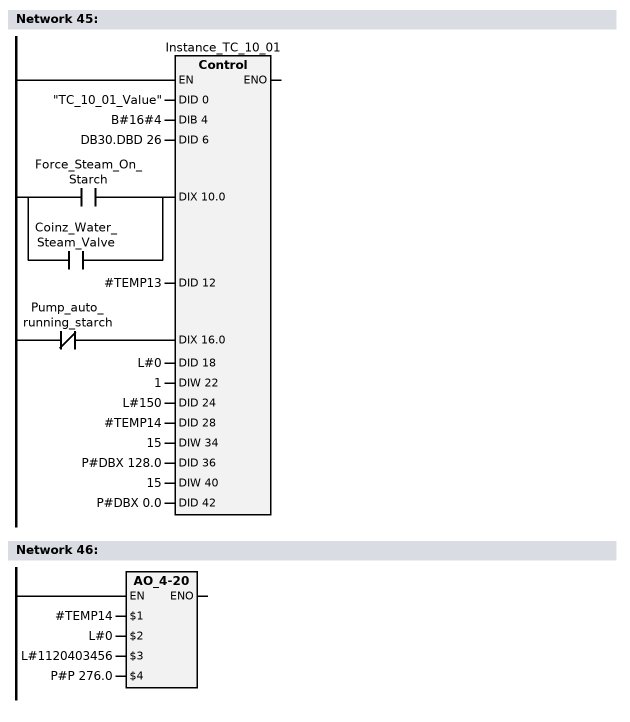
NETWORK
TITLE =
      A(;
      O     "Force_Steam_On_Starch";
      O     "Coinz_Water_Steam_Valve";
      );
      =     L 56.0;
      BLD   103;
      AN    "Pump_auto_running_starch";
      =     L 56.1;
      BLD   103;
      CALL  "Control" , "Instance_TC_10_01" (
           DID 0                    := "TC_10_01_Value",
           DIB 4                    := B#16#4,
           DID 6                    := DB30.DBD 26,
           DIX 10.0                 := L 56.0,
           DID 12                   := #TEMP13,
           DIX 16.0                 := L 56.1,
           DID 18                   := L#0,
           DIW 22                   := 1,
           DID 24                   := L#150,
           DID 28                   := #TEMP14,
           DIW 34                   := 15,
           DID 36                   := P#DBX 128.0,
           DIW 40                   := 15,
           DID 42                   := P#DBX 0.0);
      NOP   0;
NETWORK
TITLE =
      CALL  "AO_4-20" (
           $1                       := #TEMP14,
           $2                       := L#0,
           $3                       := L#1120403456,
           $4                       := P#P 276.0);
      NOP   0;
END_FUNCTION_BLOCK

FUNCTION_BLOCK "ALARM_HANDLING_STARCH"	// FB 31
AUTHOR : GAW-LK
FAMILY : ALARM
NAME : ALARMS
VERSION : 0.1
BEGIN
// (block stored without names or comments; labels and parameter names are numbered)
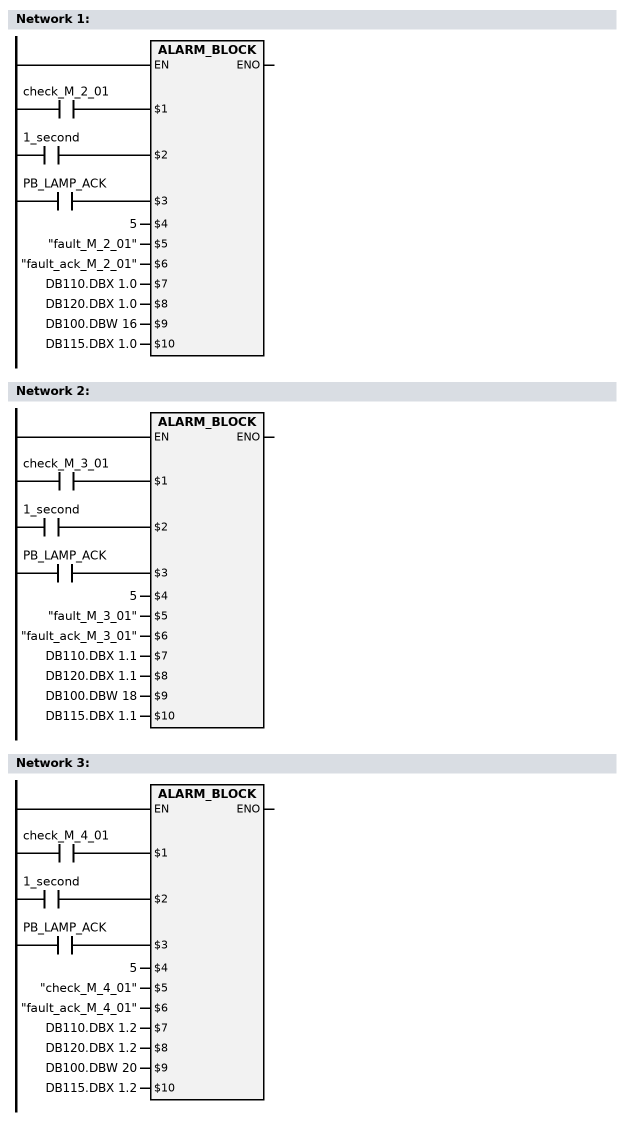
NETWORK
TITLE =
      A     "check_M_2_01";
      =     L 0.0;
      BLD   103;
      A     "1_second";
      =     L 0.1;
      BLD   103;
      A     "PB_LAMP_ACK";
      =     L 0.2;
      BLD   103;
      CALL  "ALARM_BLOCK" (
           $1                       := L 0.0,
           $2                       := L 0.1,
           $3                       := L 0.2,
           $4                       := 5,
           $5                       := "fault_M_2_01",
           $6                       := "fault_ack_M_2_01",
           $7                       := DB110.DBX 1.0,
           $8                       := DB120.DBX 1.0,
           $9                       := DB100.DBW 16,
           $10                      := DB115.DBX 1.0);
      NOP   0;
NETWORK
TITLE =
      A     "check_M_3_01";
      =     L 0.0;
      BLD   103;
      A     "1_second";
      =     L 0.1;
      BLD   103;
      A     "PB_LAMP_ACK";
      =     L 0.2;
      BLD   103;
      CALL  "ALARM_BLOCK" (
           $1                       := L 0.0,
           $2                       := L 0.1,
           $3                       := L 0.2,
           $4                       := 5,
           $5                       := "fault_M_3_01",
           $6                       := "fault_ack_M_3_01",
           $7                       := DB110.DBX 1.1,
           $8                       := DB120.DBX 1.1,
           $9                       := DB100.DBW 18,
           $10                      := DB115.DBX 1.1);
      NOP   0;
NETWORK
TITLE =
      A     "check_M_4_01";
      =     L 0.0;
      BLD   103;
      A     "1_second";
      =     L 0.1;
      BLD   103;
      A     "PB_LAMP_ACK";
      =     L 0.2;
      BLD   103;
      CALL  "ALARM_BLOCK" (
           $1                       := L 0.0,
           $2                       := L 0.1,
           $3                       := L 0.2,
           $4                       := 5,
           $5                       := "check_M_4_01",
           $6                       := "fault_ack_M_4_01",
           $7                       := DB110.DBX 1.2,
           $8                       := DB120.DBX 1.2,
           $9                       := DB100.DBW 20,
           $10                      := DB115.DBX 1.2);
      NOP   0;
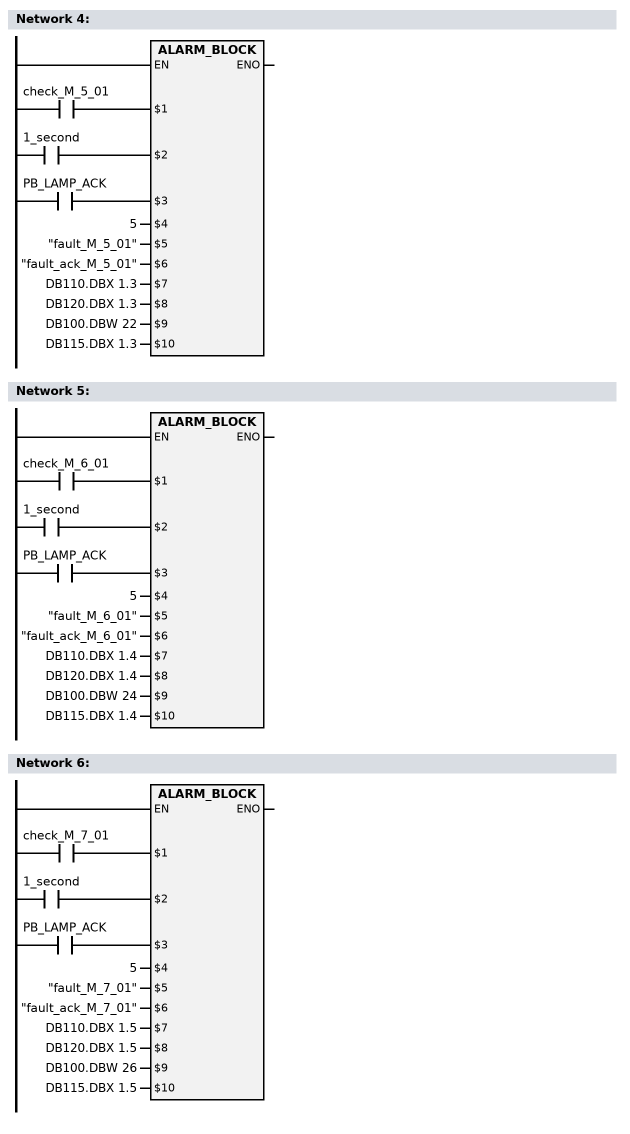
NETWORK
TITLE =
      A     "check_M_5_01";
      =     L 0.0;
      BLD   103;
      A     "1_second";
      =     L 0.1;
      BLD   103;
      A     "PB_LAMP_ACK";
      =     L 0.2;
      BLD   103;
      CALL  "ALARM_BLOCK" (
           $1                       := L 0.0,
           $2                       := L 0.1,
           $3                       := L 0.2,
           $4                       := 5,
           $5                       := "fault_M_5_01",
           $6                       := "fault_ack_M_5_01",
           $7                       := DB110.DBX 1.3,
           $8                       := DB120.DBX 1.3,
           $9                       := DB100.DBW 22,
           $10                      := DB115.DBX 1.3);
      NOP   0;
NETWORK
TITLE =
      A     "check_M_6_01";
      =     L 0.0;
      BLD   103;
      A     "1_second";
      =     L 0.1;
      BLD   103;
      A     "PB_LAMP_ACK";
      =     L 0.2;
      BLD   103;
      CALL  "ALARM_BLOCK" (
           $1                       := L 0.0,
           $2                       := L 0.1,
           $3                       := L 0.2,
           $4                       := 5,
           $5                       := "fault_M_6_01",
           $6                       := "fault_ack_M_6_01",
           $7                       := DB110.DBX 1.4,
           $8                       := DB120.DBX 1.4,
           $9                       := DB100.DBW 24,
           $10                      := DB115.DBX 1.4);
      NOP   0;
NETWORK
TITLE =
      A     "check_M_7_01";
      =     L 0.0;
      BLD   103;
      A     "1_second";
      =     L 0.1;
      BLD   103;
      A     "PB_LAMP_ACK";
      =     L 0.2;
      BLD   103;
      CALL  "ALARM_BLOCK" (
           $1                       := L 0.0,
           $2                       := L 0.1,
           $3                       := L 0.2,
           $4                       := 5,
           $5                       := "fault_M_7_01",
           $6                       := "fault_ack_M_7_01",
           $7                       := DB110.DBX 1.5,
           $8                       := DB120.DBX 1.5,
           $9                       := DB100.DBW 26,
           $10                      := DB115.DBX 1.5);
      NOP   0;
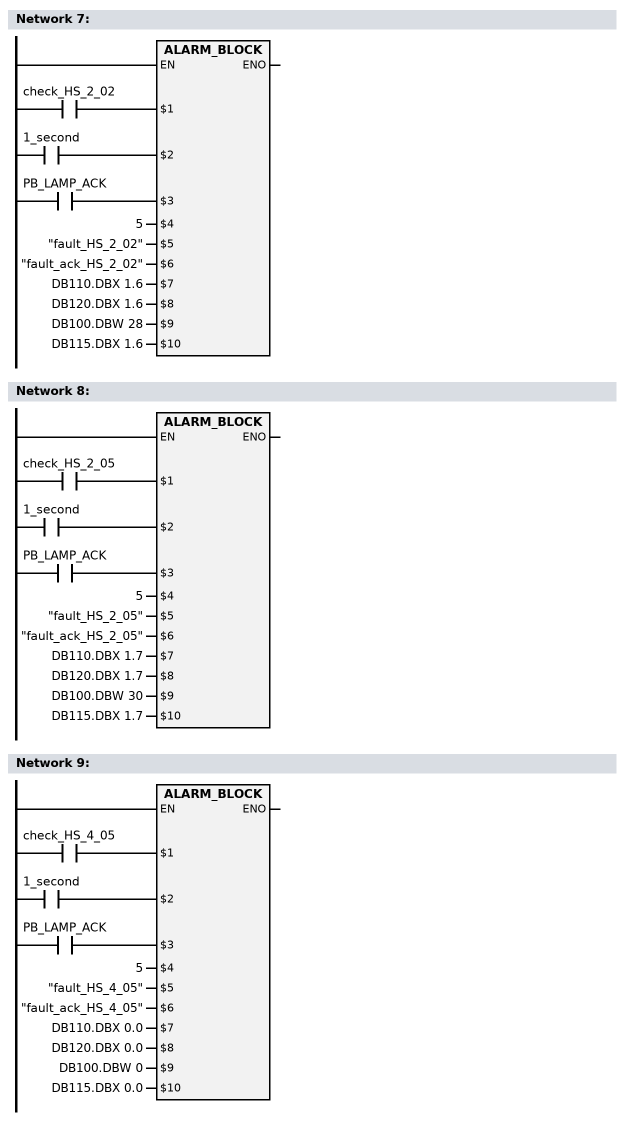
NETWORK
TITLE =
      A     "check_HS_2_02";
      =     L 0.0;
      BLD   103;
      A     "1_second";
      =     L 0.1;
      BLD   103;
      A     "PB_LAMP_ACK";
      =     L 0.2;
      BLD   103;
      CALL  "ALARM_BLOCK" (
           $1                       := L 0.0,
           $2                       := L 0.1,
           $3                       := L 0.2,
           $4                       := 5,
           $5                       := "fault_HS_2_02",
           $6                       := "fault_ack_HS_2_02",
           $7                       := DB110.DBX 1.6,
           $8                       := DB120.DBX 1.6,
           $9                       := DB100.DBW 28,
           $10                      := DB115.DBX 1.6);
      NOP   0;
NETWORK
TITLE =
      A     "check_HS_2_05";
      =     L 0.0;
      BLD   103;
      A     "1_second";
      =     L 0.1;
      BLD   103;
      A     "PB_LAMP_ACK";
      =     L 0.2;
      BLD   103;
      CALL  "ALARM_BLOCK" (
           $1                       := L 0.0,
           $2                       := L 0.1,
           $3                       := L 0.2,
           $4                       := 5,
           $5                       := "fault_HS_2_05",
           $6                       := "fault_ack_HS_2_05",
           $7                       := DB110.DBX 1.7,
           $8                       := DB120.DBX 1.7,
           $9                       := DB100.DBW 30,
           $10                      := DB115.DBX 1.7);
      NOP   0;
NETWORK
TITLE =
      A     "check_HS_4_05";
      =     L 0.0;
      BLD   103;
      A     "1_second";
      =     L 0.1;
      BLD   103;
      A     "PB_LAMP_ACK";
      =     L 0.2;
      BLD   103;
      CALL  "ALARM_BLOCK" (
           $1                       := L 0.0,
           $2                       := L 0.1,
           $3                       := L 0.2,
           $4                       := 5,
           $5                       := "fault_HS_4_05",
           $6                       := "fault_ack_HS_4_05",
           $7                       := DB110.DBX 0.0,
           $8                       := DB120.DBX 0.0,
           $9                       := DB100.DBW 0,
           $10                      := DB115.DBX 0.0);
      NOP   0;
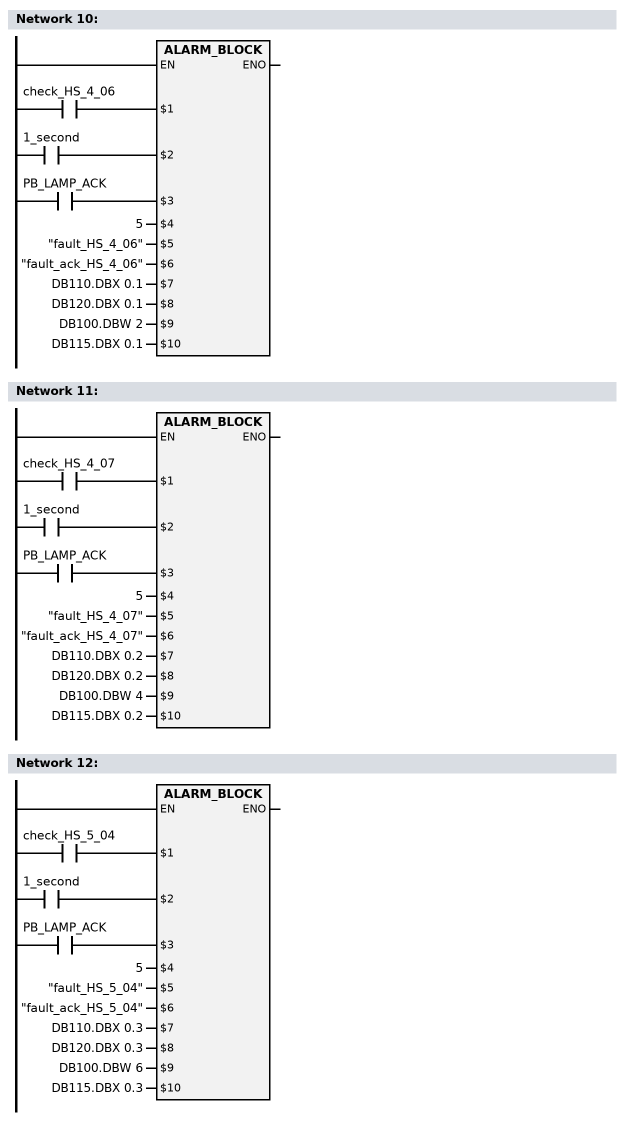
NETWORK
TITLE =
      A     "check_HS_4_06";
      =     L 0.0;
      BLD   103;
      A     "1_second";
      =     L 0.1;
      BLD   103;
      A     "PB_LAMP_ACK";
      =     L 0.2;
      BLD   103;
      CALL  "ALARM_BLOCK" (
           $1                       := L 0.0,
           $2                       := L 0.1,
           $3                       := L 0.2,
           $4                       := 5,
           $5                       := "fault_HS_4_06",
           $6                       := "fault_ack_HS_4_06",
           $7                       := DB110.DBX 0.1,
           $8                       := DB120.DBX 0.1,
           $9                       := DB100.DBW 2,
           $10                      := DB115.DBX 0.1);
      NOP   0;
NETWORK
TITLE =
      A     "check_HS_4_07";
      =     L 0.0;
      BLD   103;
      A     "1_second";
      =     L 0.1;
      BLD   103;
      A     "PB_LAMP_ACK";
      =     L 0.2;
      BLD   103;
      CALL  "ALARM_BLOCK" (
           $1                       := L 0.0,
           $2                       := L 0.1,
           $3                       := L 0.2,
           $4                       := 5,
           $5                       := "fault_HS_4_07",
           $6                       := "fault_ack_HS_4_07",
           $7                       := DB110.DBX 0.2,
           $8                       := DB120.DBX 0.2,
           $9                       := DB100.DBW 4,
           $10                      := DB115.DBX 0.2);
      NOP   0;
NETWORK
TITLE =
      A     "check_HS_5_04";
      =     L 0.0;
      BLD   103;
      A     "1_second";
      =     L 0.1;
      BLD   103;
      A     "PB_LAMP_ACK";
      =     L 0.2;
      BLD   103;
      CALL  "ALARM_BLOCK" (
           $1                       := L 0.0,
           $2                       := L 0.1,
           $3                       := L 0.2,
           $4                       := 5,
           $5                       := "fault_HS_5_04",
           $6                       := "fault_ack_HS_5_04",
           $7                       := DB110.DBX 0.3,
           $8                       := DB120.DBX 0.3,
           $9                       := DB100.DBW 6,
           $10                      := DB115.DBX 0.3);
      NOP   0;
